KUKA KRL program: MyProgram_172().src

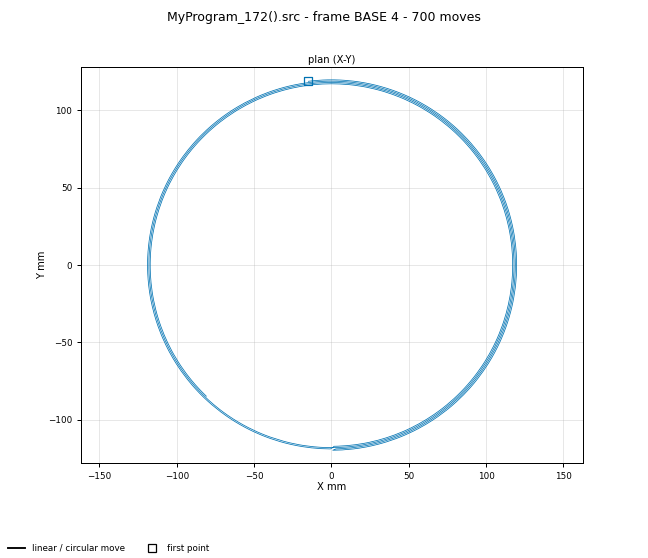
[picture p0: tool path of MyProgram_172().src in frame BASE 4, 700 of 700 moves have a stored position in this frame; points joined in program order, loops and branches not executed]
&ACCESS RVP
&REL 1
&PARAM TEMPLATE = C:\KRC\Roboter\Template\vorgabe
&PARAM EDITMASK = *
DEF MyProgram_172()
; ---- Setting reference (Base) ----
$BASE = BASE_DATA[4]

; --------------------------
; ---- Setting tool (TCP) ----
$TOOL = TOOL_DATA[3]
; --------------------------

$VEL.CP = VEL_APROX_PRINT
Startdeposition()
$VEL.CP = VEL_PRINT
LIN {X -14.9345,Y 118.8395,Z 128,A 91.9822,B 24.9419,C -1.7603,E1 24.9831,E2 354.1714} C_DIS
LIN {X -10.7622,Y 119.2891,Z 128,A 90.661,B 24.9398,C -1.7917,E1 24.9865,E2 355.4188} C_DIS
LIN {X -5.4739,Y 119.6487,Z 128,A 88.2073,B 24.9395,C -1.7964,E1 24.9934,E2 357.8622} C_DIS
LIN {X -2.3345,Y 119.7507,Z 128,A 85.9891,B 24.9416,C -1.7648,E1 24.9997,E2 360.1555} C_DIS
LIN {X 1.6856,Y 119.7625,Z 128,A 84.4618,B 24.9404,C -1.7828,E1 25.0039,E2 361.6401} C_DIS
LIN {X 5.7094,Y 119.6385,Z 128,A 82.6922,B 24.9399,C -1.7899,E1 25.0088,E2 363.3922} C_DIS
LIN {X 8.3372,Y 119.4831,Z 128,A 81.3395,B 24.9402,C -1.7857,E1 25.0126,E2 364.7544} C_DIS
LIN {X 14.2008,Y 118.9288,Z 128,A 78.7621,B 24.9395,C -1.7962,E1 25.0197,E2 367.3053} C_DIS
LIN {X 17.7257,Y 118.4559,Z 128,A 76.9686,B 24.9398,C -1.7916,E1 25.0247,E2 369.1083} C_DIS
LIN {X 21.7971,Y 117.7748,Z 128,A 74.9308,B 24.9401,C -1.788,E1 25.0303,E2 371.1525} C_DIS
LIN {X 25.2622,Y 117.0792,Z 128,A 73.1853,B 24.9403,C -1.7847,E1 25.0351,E2 372.9034} C_DIS
LIN {X 28.7779,Y 116.2654,Z 128,A 71.5409,B 24.9401,C -1.7875,E1 25.0395,E2 374.539} C_DIS
LIN {X 31.5389,Y 115.5467,Z 128,A 69.4789,B 24.9423,C -1.7548,E1 25.0453,E2 376.6751} C_DIS
LIN {X 35.9866,Y 114.2406,Z 128,A 67.9927,B 24.9402,C -1.7864,E1 25.049,E2 378.0836} C_DIS
LIN {X 39.7103,Y 112.9989,Z 128,A 65.8502,B 24.9411,C -1.7726,E1 25.0548,E2 380.2546} C_DIS
LIN {X 43.3363,Y 111.6596,Z 128,A 63.849,B 24.9417,C -1.7638,E1 25.06,E2 382.2724} C_DIS
LIN {X 47.456,Y 109.9717,Z 128,A 61.9358,B 24.9412,C -1.7715,E1 25.0649,E2 384.163} C_DIS
LIN {X 50.5894,Y 108.565,Z 128,A 60.3762,B 24.9411,C -1.7734,E1 25.0688,E2 385.714} C_DIS
LIN {X 54.0331,Y 106.8942,Z 128,A 58.4921,B 24.9414,C -1.7686,E1 25.0735,E2 387.6044} C_DIS
LIN {X 57.312,Y 105.1715,Z 128,A 56.7697,B 24.9414,C -1.7685,E1 25.0778,E2 389.3222} C_DIS
LIN {X 61.1307,Y 102.9987,Z 128,A 54.6582,B 24.9416,C -1.765,E1 25.0829,E2 391.4356} C_DIS
LIN {X 64.4896,Y 100.9297,Z 128,A 52.5109,B 24.9426,C -1.7498,E1 25.088,E2 393.6118} C_DIS
LIN {X 69.9469,Y 97.2281,Z 128,A 49.8821,B 24.9413,C -1.7692,E1 25.0939,E2 396.1859} C_DIS
LIN {X 73.3681,Y 94.6725,Z 128,A 47.6716,B 24.9421,C -1.7576,E1 25.0989,E2 398.4159} C_DIS
LIN {X 76.4144,Y 92.2308,Z 128,A 45.7857,B 24.9424,C -1.7531,E1 25.103,E2 400.3051} C_DIS
LIN {X 78.8231,Y 90.1808,Z 128,A 44.2978,B 24.9425,C -1.7513,E1 25.1061,E2 401.7914} C_DIS
LIN {X 81.4658,Y 87.8033,Z 128,A 42.4667,B 24.9432,C -1.7416,E1 25.11,E2 403.638} C_DIS
LIN {X 84.2691,Y 85.114,Z 128,A 40.7422,B 24.943,C -1.744,E1 25.1134,E2 405.3497} C_DIS
LIN {X 88.0039,Y 81.2472,Z 128,A 38.3973,B 24.9427,C -1.7491,E1 25.1179,E2 407.6724} C_DIS
LIN {X 90.3573,Y 78.621,Z 128,A 36.5475,B 24.9434,C -1.7374,E1 25.1213,E2 409.5416} C_DIS
LIN {X 93.9931,Y 74.2358,Z 128,A 33.8716,B 24.9437,C -1.7332,E1 25.1261,E2 412.2149} C_DIS
LIN {X 95.9007,Y 71.7548,Z 128,A 32.2244,B 24.9444,C -1.7223,E1 25.1289,E2 413.88} C_DIS
LIN {X 98.383,Y 68.3114,Z 128,A 30.2874,B 24.9444,C -1.7216,E1 25.132,E2 415.8092} C_DIS
LIN {X 100.4183,Y 65.2864,Z 128,A 28.4483,B 24.945,C -1.7125,E1 25.1348,E2 417.6608} C_DIS
LIN {X 102.3996,Y 62.1288,Z 128,A 26.0566,B 24.9472,C -1.6786,E1 25.1384,E2 420.1201} C_DIS
LIN {X 104.9804,Y 57.6644,Z 128,A 24.2184,B 24.9457,C -1.7019,E1 25.1408,E2 421.8939} C_DIS
LIN {X 106.7304,Y 54.3535,Z 128,A 22.5591,B 24.9457,C -1.7032,E1 25.1429,E2 423.5412} C_DIS
LIN {X 108.2379,Y 51.2896,Z 128,A 20.9731,B 24.9457,C -1.7009,E1 25.1449,E2 425.1243} C_DIS
LIN {X 109.6146,Y 48.2751,Z 128,A 19.0189,B 24.9472,C -1.6784,E1 25.1471,E2 427.1208} C_DIS
LIN {X 111.6551,Y 43.3476,Z 128,A 16.4448,B 24.9478,C -1.6698,E1 25.1498,E2 429.7011} C_DIS
LIN {X 112.8514,Y 40.1306,Z 128,A 15.3331,B 24.9464,C -1.6905,E1 25.1508,E2 430.7575} C_DIS
LIN {X 114.185,Y 36.1643,Z 128,A 13.0854,B 24.9476,C -1.6725,E1 25.1528,E2 433.0351} C_DIS
LIN {X 115.1759,Y 32.8666,Z 128,A 11.4964,B 24.9477,C -1.6702,E1 25.154,E2 434.6203} C_DIS
LIN {X 116.2749,Y 28.739,Z 128,A 9.4821,B 24.948,C -1.6653,E1 25.1554,E2 436.6346} C_DIS
LIN {X 117.0488,Y 25.4019,Z 128,A 7.9707,B 24.948,C -1.6664,E1 25.1563,E2 438.1348} C_DIS
LIN {X 117.6341,Y 22.5364,Z 128,A 6.5322,B 24.9484,C -1.66,E1 25.1571,E2 439.5799} C_DIS
LIN {X 118.2492,Y 19.0601,Z 128,A 4.6721,B 24.9492,C -1.6462,E1 25.158,E2 441.4616} C_DIS
LIN {X 119.1222,Y 12.4724,Z 128,A 2.0396,B 24.9482,C -1.6628,E1 25.1589,E2 444.0394} C_DIS
LIN {X 119.5152,Y 7.8623,Z 128,A -0.5581,B 24.9498,C -1.6367,E1 25.1595,E2 446.6832} C_DIS
LIN {X 119.7603,Y 1.8102,Z 128,A -3.0517,B 24.9492,C -1.6471,E1 25.1598,E2 449.1375} C_DIS
LIN {X 119.7522,Y -2.2507,Z 128,A -5.9251,B 24.9523,C -1.5952,E1 25.1597,E2 452.1161} C_DIS
LIN {X 119.5842,Y -6.7302,Z 128,A -7.1659,B 24.9501,C -1.6323,E1 25.1595,E2 453.2621} C_DIS
LIN {X 119.1569,Y -12.1411,Z 128,A -9.8149,B 24.9508,C -1.6211,E1 25.159,E2 455.9217} C_DIS
LIN {X 118.8189,Y -15.0932,Z 128,A -12.4654,B 24.9546,C -1.5566,E1 25.158,E2 458.7086} C_DIS
LIN {X 117.8363,Y -21.4551,Z 128,A -14.3715,B 24.9518,C -1.6036,E1 25.1571,E2 460.4928} C_DIS
LIN {X 117.3034,Y -24.199,Z 128,A -15.8035,B 24.9524,C -1.5946,E1 25.1563,E2 461.9377} C_DIS
LIN {X 116.6602,Y -27.131,Z 128,A -17.1963,B 24.9525,C -1.5921,E1 25.1555,E2 463.3283} C_DIS
LIN {X 115.915,Y -30.1577,Z 128,A -18.8453,B 24.9533,C -1.5795,E1 25.1543,E2 464.9974} C_DIS
LIN {X 114.8429,Y -34.0113,Z 128,A -20.6089,B 24.9532,C -1.5807,E1 25.153,E2 466.7481} C_DIS
LIN {X 113.9274,Y -36.9624,Z 128,A -22.1194,B 24.9536,C -1.5744,E1 25.1517,E2 468.2649} C_DIS
LIN {X 112.6185,Y -40.7776,Z 128,A -23.9811,B 24.9537,C -1.5716,E1 25.15,E2 470.1227} C_DIS
LIN {X 111.418,Y -43.9513,Z 128,A -25.65,B 24.9542,C -1.5643,E1 25.1483,E2 471.7995} C_DIS
LIN {X 109.366,Y -48.8355,Z 128,A -27.9679,B 24.954,C -1.567,E1 25.1458,E2 474.0982} C_DIS
LIN {X 107.4011,Y -53.0161,Z 128,A -30.0733,B 24.954,C -1.5654,E1 25.1433,E2 476.1962} C_DIS
LIN {X 105.5247,Y -56.6608,Z 128,A -32.7446,B 24.9564,C -1.5248,E1 25.1397,E2 478.9491} C_DIS
LIN {X 103.7146,Y -59.9083,Z 128,A -33.6102,B 24.9542,C -1.5641,E1 25.1386,E2 479.7175} C_DIS
LIN {X 101.3114,Y -63.8899,Z 128,A -36.3268,B 24.9559,C -1.5335,E1 25.1346,E2 482.4925} C_DIS
LIN {X 98.3282,Y -68.3902,Z 128,A -38.6382,B 24.9556,C -1.5394,E1 25.1311,E2 484.7785} C_DIS
LIN {X 94.2998,Y -73.8478,Z 128,A -42.0752,B 24.9567,C -1.521,E1 25.1253,E2 488.2423} C_DIS
LIN {X 92.1735,Y -76.4833,Z 128,A -44.2995,B 24.9585,C -1.4875,E1 25.1212,E2 490.5355} C_DIS
LIN {X 89.1898,Y -79.9427,Z 128,A -46.6277,B 24.9592,C -1.475,E1 25.1168,E2 492.8828} C_DIS
LIN {X 85.5452,Y -83.8326,Z 128,A -48.3712,B 24.9574,C -1.5074,E1 25.1136,E2 494.5425} C_DIS
LIN {X 80.5462,Y -88.6471,Z 128,A -52.2709,B 24.9594,C -1.4715,E1 25.1055,E2 498.5108} C_DIS
LIN {X 77.2653,Y -91.5206,Z 128,A -53.8492,B 24.9584,C -1.491,E1 25.1023,E2 500.0369} C_DIS
LIN {X 74.2886,Y -93.9514,Z 128,A -56.7192,B 24.9613,C -1.4379,E1 25.0958,E2 503.0217} C_DIS
LIN {X 68.7364,Y -98.0875,Z 128,A -58.7295,B 24.9583,C -1.4928,E1 25.0915,E2 504.8953} C_DIS
LIN {X 65.3681,Y -100.3649,Z 128,A -61.6332,B 24.961,C -1.4433,E1 25.0845,E2 507.9063} C_DIS
LIN {X 60.8442,Y -103.1681,Z 128,A -62.9572,B 24.958,C -1.4966,E1 25.0816,E2 509.1002} C_DIS
LIN {X 55.6149,Y -106.0787,Z 128,A -66.1813,B 24.9593,C -1.4741,E1 25.0736,E2 512.368} C_DIS
LIN {X 52.8498,Y -107.4835,Z 128,A -67.6815,B 24.9595,C -1.4708,E1 25.0699,E2 513.8719} C_DIS
LIN {X 47.3838,Y -110.0032,Z 128,A -70.4733,B 24.9595,C -1.4705,E1 25.0628,E2 516.6576} C_DIS
LIN {X 44.9683,Y -111.0115,Z 128,A -71.7797,B 24.9597,C -1.4661,E1 25.0594,E2 517.9713} C_DIS
LIN {X 41.9329,Y -112.1943,Z 128,A -74.48,B 24.9627,C -1.4105,E1 25.052,E2 520.7973} C_DIS
LIN {X 35.5057,Y -114.3897,Z 128,A -76.5649,B 24.96,C -1.4608,E1 25.0468,E2 522.7594} C_DIS
LIN {X 32.4814,Y -115.2851,Z 128,A -78.0718,B 24.9601,C -1.4592,E1 25.0427,E2 524.2676} C_DIS
LIN {X 29.6802,Y -116.0378,Z 128,A -79.4968,B 24.9603,C -1.456,E1 25.0389,E2 525.698} C_DIS
LIN {X 25.968,Y -116.9253,Z 128,A -81.4039,B 24.9606,C -1.4504,E1 25.0336,E2 527.6156} C_DIS
LIN {X 22.512,Y -117.6388,Z 128,A -83.6176,B 24.962,C -1.4246,E1 25.0274,E2 529.8878} C_DIS
LIN {X 18.0591,Y -118.4043,Z 128,A -85.6229,B 24.9617,C -1.4302,E1 25.0219,E2 531.878} C_DIS
LIN {X 14.2771,Y -118.9199,Z 128,A -86.9177,B 24.9604,C -1.4536,E1 25.0185,E2 533.1163} C_DIS
LIN {X 6.9052,Y -119.5745,Z 128,A -90.2911,B 24.9601,C -1.4595,E1 25.0092,E2 536.4739} C_DIS
LIN {X 0.8345,Y -119.7701,Z 128,A -93.2214,B 24.9602,C -1.4573,E1 25.001,E2 539.4087} C_DIS
Enddeposition()
LIN {X 0.8345,Y -119.7701,Z 128,A -93.2214,B 24.9602,C -1.4573,E1 25.001,E2 539.4087} C_DIS
Startdeposition()
$VEL.CP = VEL_PRINT
LIN {X 2.8953,Y -118.8882,Z 128,A -91.2381,B 24.9568,C -1.5184,E1 25.0069,E2 537.281} C_DIS
LIN {X 6.7932,Y -118.7278,Z 128,A -89.9008,B 24.9582,C -1.4939,E1 25.0105,E2 536.0023} C_DIS
LIN {X 12.3059,Y -118.2834,Z 128,A -87.272,B 24.9582,C -1.4936,E1 25.0178,E2 533.3757} C_DIS
LIN {X 15.4448,Y -117.9146,Z 128,A -85.7393,B 24.9582,C -1.495,E1 25.022,E2 531.8408} C_DIS
LIN {X 17.8503,Y -117.5749,Z 128,A -84.5445,B 24.958,C -1.497,E1 25.0253,E2 530.6425} C_DIS
LIN {X 23.2009,Y -116.6389,Z 128,A -81.8074,B 24.9576,C -1.5047,E1 25.0329,E2 527.8902} C_DIS
LIN {X 26.8874,Y -115.8424,Z 128,A -80.0744,B 24.9577,C -1.5025,E1 25.0376,E2 526.1647} C_DIS
LIN {X 30.6338,Y -114.9091,Z 128,A -78.1946,B 24.9575,C -1.5053,E1 25.0427,E2 524.281} C_DIS
LIN {X 33.7472,Y -114.0329,Z 128,A -76.6918,B 24.9575,C -1.5045,E1 25.0467,E2 522.7828} C_DIS
LIN {X 39.8877,Y -112.0341,Z 128,A -73.4398,B 24.957,C -1.515,E1 25.0554,E2 519.5121} C_DIS
LIN {X 43.5273,Y -110.6696,Z 128,A -71.7253,B 24.9573,C -1.5101,E1 25.0598,E2 517.813} C_DIS
LIN {X 46.4605,Y -109.471,Z 128,A -70.0701,B 24.9568,C -1.5185,E1 25.0641,E2 516.1419} C_DIS
LIN {X 49.1217,Y -108.3029,Z 128,A -68.4485,B 24.9561,C -1.5313,E1 25.0683,E2 514.4941} C_DIS
LIN {X 52.1685,Y -106.8707,Z 128,A -67.0331,B 24.9565,C -1.524,E1 25.0718,E2 513.0997} C_DIS
LIN {X 55.0721,Y -105.4021,Z 128,A -65.0797,B 24.9553,C -1.5453,E1 25.0768,E2 511.1014} C_DIS
LIN {X 58.7314,Y -103.4087,Z 128,A -63.5195,B 24.9563,C -1.5273,E1 25.0804,E2 509.5883} C_DIS
LIN {X 61.3868,Y -101.854,Z 128,A -61.5561,B 24.9548,C -1.5533,E1 25.0853,E2 507.5695} C_DIS
LIN {X 65.0646,Y -99.545,Z 128,A -60.0756,B 24.9563,C -1.5278,E1 25.0886,E2 506.154} C_DIS
LIN {X 67.6195,Y -97.8268,Z 128,A -58.7214,B 24.9564,C -1.5246,E1 25.0917,E2 504.812} C_DIS
LIN {X 72.6114,Y -94.1805,Z 128,A -55.5369,B 24.9555,C -1.5409,E1 25.0989,E2 501.6005} C_DIS
LIN {X 75.9071,Y -91.5451,Z 128,A -53.5631,B 24.9555,C -1.5426,E1 25.1031,E2 499.6301} C_DIS
LIN {X 78.1001,Y -89.6816,Z 128,A -51.9193,B 24.9545,C -1.5583,E1 25.1067,E2 497.9558} C_DIS
LIN {X 83.0665,Y -85.1049,Z 128,A -48.8714,B 24.9546,C -1.5561,E1 25.1128,E2 494.9257} C_DIS
LIN {X 85.6964,Y -82.4532,Z 128,A -47.4083,B 24.9553,C -1.5442,E1 25.1156,E2 493.4967} C_DIS
LIN {X 88.759,Y -79.1471,Z 128,A -44.6852,B 24.9534,C -1.5767,E1 25.1209,E2 490.709} C_DIS
LIN {X 90.922,Y -76.6547,Z 128,A -43.3461,B 24.9539,C -1.5686,E1 25.1232,E2 489.3952} C_DIS
LIN {X 93.1098,Y -73.9801,Z 128,A -41.8006,B 24.9539,C -1.5673,E1 25.1259,E2 487.86} C_DIS
LIN {X 96.737,Y -69.1689,Z 128,A -39.2022,B 24.9544,C -1.5604,E1 25.1302,E2 485.2902} C_DIS
LIN {X 98.2379,Y -67.0214,Z 128,A -37.4167,B 24.9527,C -1.5895,E1 25.1332,E2 483.4448} C_DIS
LIN {X 100.7124,Y -63.2414,Z 128,A -35.2399,B 24.9523,C -1.5958,E1 25.1364,E2 481.2641} C_DIS
LIN {X 103.0299,Y -59.3906,Z 128,A -33.3725,B 24.9528,C -1.5875,E1 25.139,E2 479.4259} C_DIS
LIN {X 105.3544,Y -55.1625,Z 128,A -30.927,B 24.952,C -1.6004,E1 25.1423,E2 476.9628} C_DIS
LIN {X 107.6576,Y -50.5209,Z 128,A -28.5211,B 24.9518,C -1.6035,E1 25.1452,E2 474.5625} C_DIS
LIN {X 109.3932,Y -46.6451,Z 128,A -26.3521,B 24.9511,C -1.6159,E1 25.1477,E2 472.3762} C_DIS
LIN {X 111.054,Y -42.5393,Z 128,A -24.3086,B 24.9509,C -1.6181,E1 25.1498,E2 470.3387} C_DIS
LIN {X 112.2755,Y -39.1998,Z 128,A -22.6928,B 24.9509,C -1.6187,E1 25.1513,E2 468.7306} C_DIS
LIN {X 113.4977,Y -35.5069,Z 128,A -20.8268,B 24.9506,C -1.6243,E1 25.1529,E2 466.862} C_DIS
LIN {X 114.4075,Y -32.4548,Z 128,A -19.3213,B 24.9504,C -1.6278,E1 25.154,E2 465.3569} C_DIS
LIN {X 115.2334,Y -29.3887,Z 128,A -17.7706,B 24.95,C -1.6337,E1 25.1551,E2 463.8011} C_DIS
LIN {X 116.1074,Y -25.7218,Z 128,A -15.9405,B 24.9496,C -1.6403,E1 25.1563,E2 461.9662} C_DIS
LIN {X 116.8616,Y -22.0444,Z 128,A -14.2309,B 24.9496,C -1.6413,E1 25.1572,E2 460.2643} C_DIS
LIN {X 117.8335,Y -16.0654,Z 128,A -11.1596,B 24.9485,C -1.6583,E1 25.1585,E2 457.1709} C_DIS
LIN {X 118.2758,Y -12.3783,Z 128,A -9.5565,B 24.9487,C -1.655,E1 25.159,E2 455.585} C_DIS
LIN {X 118.6721,Y -7.7074,Z 128,A -7.3093,B 24.9482,C -1.6618,E1 25.1595,E2 453.335} C_DIS
LIN {X 118.876,Y -3.3144,Z 128,A -5.0425,B 24.9474,C -1.6761,E1 25.1598,E2 451.0482} C_DIS
LIN {X 118.9205,Y 0.6044,Z 128,A -3.1956,B 24.9471,C -1.6802,E1 25.1598,E2 449.2025} C_DIS
LIN {X 118.8667,Y 3.6165,Z 128,A -1.6079,B 24.9464,C -1.6917,E1 25.1596,E2 447.5972} C_DIS
LIN {X 118.671,Y 7.7236,Z 128,A 0.2246,B 24.9464,C -1.6908,E1 25.1594,E2 445.7777} C_DIS
LIN {X 118.3124,Y 12.0286,Z 128,A 2.1778,B 24.9464,C -1.6912,E1 25.1589,E2 443.8351} C_DIS
LIN {X 117.7508,Y 16.6472,Z 128,A 4.5059,B 24.9457,C -1.7027,E1 25.158,E2 441.4937} C_DIS
LIN {X 117.1261,Y 20.5928,Z 128,A 6.365,B 24.9455,C -1.7056,E1 25.1572,E2 439.6387} C_DIS
LIN {X 116.5594,Y 23.5879,Z 128,A 7.8405,B 24.9452,C -1.7106,E1 25.1564,E2 438.1599} C_DIS
LIN {X 115.819,Y 26.9889,Z 128,A 9.5065,B 24.9449,C -1.7153,E1 25.1553,E2 436.4925} C_DIS
LIN {X 114.8458,Y 30.8681,Z 128,A 11.422,B 24.9445,C -1.7208,E1 25.154,E2 434.5752} C_DIS
LIN {X 113.7732,Y 34.6183,Z 128,A 13.2275,B 24.9444,C -1.7229,E1 25.1526,E2 432.7749} C_DIS
LIN {X 112.7393,Y 37.8453,Z 128,A 14.874,B 24.944,C -1.7286,E1 25.1511,E2 431.1244} C_DIS
LIN {X 111.527,Y 41.2829,Z 128,A 16.9498,B 24.9426,C -1.7495,E1 25.1491,E2 429.0109} C_DIS
LIN {X 110.3497,Y 44.3353,Z 128,A 18.1014,B 24.9437,C -1.7334,E1 25.148,E2 427.9036} C_DIS
LIN {X 108.8295,Y 47.9451,Z 128,A 20.1616,B 24.9428,C -1.7473,E1 25.1457,E2 425.8219} C_DIS
LIN {X 107.237,Y 51.4063,Z 128,A 21.7999,B 24.9431,C -1.743,E1 25.1437,E2 424.2025} C_DIS
LIN {X 105.9398,Y 54.0291,Z 128,A 23.2433,B 24.9427,C -1.7486,E1 25.1419,E2 422.7536} C_DIS
LIN {X 104.2675,Y 57.1925,Z 128,A 25.4236,B 24.9409,C -1.7756,E1 25.139,E2 420.521} C_DIS
LIN {X 102.4918,Y 60.3147,Z 128,A 26.725,B 24.942,C -1.7595,E1 25.1372,E2 419.2645} C_DIS
LIN {X 100.7835,Y 63.1275,Z 128,A 28.3407,B 24.9416,C -1.7652,E1 25.1348,E2 417.6436} C_DIS
LIN {X 98.755,Y 66.2577,Z 128,A 30.1557,B 24.9412,C -1.7707,E1 25.132,E2 415.8245} C_DIS
LIN {X 96.2669,Y 69.8237,Z 128,A 32.2134,B 24.941,C -1.7742,E1 25.1287,E2 413.7685} C_DIS
LIN {X 94.1897,Y 72.5994,Z 128,A 34.0169,B 24.9403,C -1.7848,E1 25.1256,E2 411.9486} C_DIS
LIN {X 90.6307,Y 76.9967,Z 128,A 36.53,B 24.9405,C -1.7811,E1 25.1212,E2 409.4559} C_DIS
LIN {X 88.4803,Y 79.4585,Z 128,A 38.1178,B 24.9403,C -1.7853,E1 25.1182,E2 407.8651} C_DIS
LIN {X 85.1795,Y 82.9895,Z 128,A 40.5633,B 24.9395,C -1.7961,E1 25.1135,E2 405.4048} C_DIS
LIN {X 82.6255,Y 85.5302,Z 128,A 42.0321,B 24.9401,C -1.7871,E1 25.1106,E2 403.9634} C_DIS
LIN {X 80.4784,Y 87.5535,Z 128,A 43.5573,B 24.9396,C -1.795,E1 25.1075,E2 402.4258} C_DIS
LIN {X 77.9739,Y 89.7918,Z 128,A 45.2458,B 24.9392,C -1.8016,E1 25.1039,E2 400.7285} C_DIS
LIN {X 74.9657,Y 92.3176,Z 128,A 47.0262,B 24.9392,C -1.7999,E1 25.1001,E2 398.9588} C_DIS
LIN {X 72.7007,Y 94.1117,Z 128,A 48.4539,B 24.939,C -1.8042,E1 25.0969,E2 397.5264} C_DIS
LIN {X 69.7825,Y 96.297,Z 128,A 50.2933,B 24.9385,C -1.8112,E1 25.0928,E2 395.6768} C_DIS
LIN {X 64.2278,Y 100.0858,Z 128,A 53.4071,B 24.9385,C -1.8106,E1 25.0856,E2 392.5749} C_DIS
LIN {X 61.242,Y 101.942,Z 128,A 55.116,B 24.9383,C -1.8139,E1 25.0815,E2 390.8637} C_DIS
LIN {X 57.6928,Y 103.9906,Z 128,A 57.2015,B 24.9378,C -1.8219,E1 25.0764,E2 388.7653} C_DIS
LIN {X 53.9956,Y 105.9569,Z 128,A 59.1105,B 24.9379,C -1.8196,E1 25.0717,E2 386.8672} C_DIS
LIN {X 50.427,Y 107.7013,Z 128,A 61.0237,B 24.9378,C -1.8219,E1 25.0669,E2 384.9535} C_DIS
LIN {X 46.8967,Y 109.2865,Z 128,A 62.857,B 24.9378,C -1.8225,E1 25.0622,E2 383.1231} C_DIS
LIN {X 42.8741,Y 110.9262,Z 128,A 65.0568,B 24.9373,C -1.8296,E1 25.0565,E2 380.9115} C_DIS
LIN {X 39.952,Y 112.0116,Z 128,A 66.5498,B 24.9372,C -1.8306,E1 25.0526,E2 379.4192} C_DIS
LIN {X 36.6887,Y 113.1209,Z 128,A 68.4007,B 24.9365,C -1.8408,E1 25.0476,E2 377.5476} C_DIS
LIN {X 30.1916,Y 115.027,Z 128,A 71.4659,B 24.937,C -1.8339,E1 25.0394,E2 374.5038} C_DIS
LIN {X 26.7632,Y 115.8711,Z 128,A 73.038,B 24.9373,C -1.829,E1 25.0352,E2 372.9457} C_DIS
LIN {X 23.4752,Y 116.5826,Z 128,A 74.7218,B 24.937,C -1.8326,E1 25.0306,E2 371.2554} C_DIS
LIN {X 19.8865,Y 117.2475,Z 128,A 76.4532,B 24.937,C -1.8321,E1 25.0258,E2 369.5271} C_DIS
LIN {X 16.75,Y 117.7362,Z 128,A 78.007,B 24.937,C -1.8336,E1 25.0215,E2 367.9711} C_DIS
LIN {X 13.6908,Y 118.1311,Z 128,A 79.6517,B 24.9365,C -1.8411,E1 25.0169,E2 366.3098} C_DIS
LIN {X 9.647,Y 118.5299,Z 128,A 81.4354,B 24.937,C -1.8334,E1 25.012,E2 364.5455} C_DIS
LIN {X 6.2648,Y 118.757,Z 128,A 83.1346,B 24.9368,C -1.8364,E1 25.0072,E2 362.8399} C_DIS
LIN {X 3.5328,Y 118.8693,Z 128,A 84.6064,B 24.9363,C -1.8433,E1 25.0031,E2 361.3521} C_DIS
LIN {X -2.1225,Y 118.9028,Z 128,A 87.0611,B 24.9372,C -1.8305,E1 24.9963,E2 358.9278} C_DIS
LIN {X -5.3436,Y 118.8019,Z 128,A 88.6163,B 24.9372,C -1.8301,E1 24.992,E2 357.3732} C_DIS
LIN {X -9.9585,Y 118.505,Z 128,A 90.8353,B 24.9373,C -1.8287,E1 24.9858,E2 355.1566} C_DIS
LIN {X -14.4655,Y 118.0404,Z 128,A 93.1902,B 24.9369,C -1.8352,E1 24.9792,E2 352.7849} C_DIS
LIN {X -17.7189,Y 117.5952,Z 128,A 94.6264,B 24.9374,C -1.8276,E1 24.9753,E2 351.3654} C_DIS
LIN {X -20.0668,Y 117.2174,Z 128,A 95.9288,B 24.937,C -1.8338,E1 24.9717,E2 350.0472} C_DIS
LIN {X -23.801,Y 116.5157,Z 128,A 97.6167,B 24.9375,C -1.8259,E1 24.9671,E2 348.376} C_DIS
LIN {X -26.8424,Y 115.8528,Z 128,A 99.0777,B 24.9377,C -1.8228,E1 24.9631,E2 346.9205} C_DIS
LIN {X -30.0884,Y 115.0535,Z 128,A 100.6609,B 24.9379,C -1.82,E1 24.9588,E2 345.3417} C_DIS
LIN {X -33.5329,Y 114.0965,Z 128,A 102.5958,B 24.9374,C -1.8275,E1 24.9536,E2 343.3858} C_DIS
LIN {X -37.7675,Y 112.7655,Z 128,A 104.995,B 24.9368,C -1.8365,E1 24.9472,E2 340.9609} C_DIS
LIN {X -41.0134,Y 111.626,Z 128,A 106.5558,B 24.9372,C -1.8301,E1 24.9431,E2 339.4123} C_DIS
LIN {X -45.7223,Y 109.7821,Z 128,A 108.7756,B 24.9381,C -1.8171,E1 24.9374,E2 337.2184} C_DIS
LIN {X -48.9642,Y 108.3739,Z 128,A 110.4611,B 24.9383,C -1.8138,E1 24.9331,E2 335.5367} C_DIS
LIN {X -56.0854,Y 104.868,Z 128,A 114.2258,B 24.9389,C -1.8048,E1 24.9238,E2 331.7832} C_DIS
LIN {X -60.9352,Y 102.125,Z 128,A 117.353,B 24.938,C -1.8193,E1 24.9161,E2 328.6124} C_DIS
LIN {X -63.8798,Y 100.3092,Z 128,A 118.7133,B 24.9391,C -1.8027,E1 24.913,E2 327.2871} C_DIS
LIN {X -67.1467,Y 98.1531,Z 128,A 121.0288,B 24.9381,C -1.8176,E1 24.9075,E2 324.9284} C_DIS
LIN {X -70.3204,Y 95.9032,Z 128,A 122.4423,B 24.9397,C -1.7938,E1 24.9045,E2 323.5667} C_DIS
LIN {X -72.843,Y 94.0021,Z 128,A 124.33,B 24.9388,C -1.8063,E1 24.9002,E2 321.6424} C_DIS
LIN {X -75.5923,Y 91.8067,Z 128,A 125.7074,B 24.94,C -1.7888,E1 24.8973,E2 320.3013} C_DIS
LIN {X -78.0818,Y 89.6975,Z 128,A 127.6243,B 24.9393,C -1.8001,E1 24.8932,E2 318.35} C_DIS
LIN {X -80.735,Y 87.3181,Z 128,A 128.8408,B 24.941,C -1.7745,E1 24.8908,E2 317.1896} C_DIS
LIN {X -84.8387,Y 83.336,Z 128,A 131.8205,B 24.9408,C -1.7774,E1 24.8848,E2 314.1904} C_DIS
LIN {X -87.002,Y 81.076,Z 128,A 133.6264,B 24.9402,C -1.7864,E1 24.8813,E2 312.3552} C_DIS
LIN {X -89.3075,Y 78.5284,Z 128,A 135.6609,B 24.9394,C -1.7984,E1 24.8775,E2 310.2829} C_DIS
LIN {X -92.6334,Y 74.5761,Z 128,A 137.5207,B 24.9416,C -1.7648,E1 24.8744,E2 308.4945} C_DIS
LIN {X -95.8128,Y 70.444,Z 128,A 139.9826,B 24.9422,C -1.7558,E1 24.8702,E2 306.0423} C_DIS
LIN {X -98.1595,Y 67.1373,Z 128,A 142.1479,B 24.942,C -1.7594,E1 24.8668,E2 303.8579} C_DIS
LIN {X -100.6825,Y 63.2893,Z 128,A 143.9033,B 24.9437,C -1.7335,E1 24.8642,E2 302.1553} C_DIS
LIN {X -103.2815,Y 58.9528,Z 128,A 146.0966,B 24.9448,C -1.7162,E1 24.8611,E2 299.9918} C_DIS
LIN {X -104.8822,Y 56.0591,Z 128,A 148.3085,B 24.9434,C -1.7374,E1 24.8581,E2 297.7176} C_DIS
LIN {X -106.7832,Y 52.3451,Z 128,A 150.24,B 24.944,C -1.7281,E1 24.8556,E2 295.798} C_DIS
LIN {X -109.0275,Y 47.4908,Z 128,A 152.7832,B 24.9446,C -1.7188,E1 24.8527,E2 293.263} C_DIS
LIN {X -110.4216,Y 44.1585,Z 128,A 154.6909,B 24.9446,C -1.7204,E1 24.8507,E2 291.3408} C_DIS
LIN {X -112.9098,Y 37.3392,Z 128,A 158.1235,B 24.9454,C -1.7067,E1 24.8475,E2 287.9215} C_DIS
LIN {X -113.9717,Y 33.9538,Z 128,A 159.8185,B 24.9458,C -1.7007,E1 24.8461,E2 286.2312} C_DIS
LIN {X -114.879,Y 30.7452,Z 128,A 161.9292,B 24.9448,C -1.7168,E1 24.8446,E2 284.0696} C_DIS
LIN {X -115.8564,Y 26.8266,Z 128,A 163.3574,B 24.9466,C -1.6887,E1 24.8437,E2 282.7001} C_DIS
LIN {X -116.6289,Y 23.2493,Z 128,A 165.2692,B 24.9466,C -1.6892,E1 24.8426,E2 280.7759} C_DIS
LIN {X -117.2972,Y 19.5892,Z 128,A 166.9465,B 24.9472,C -1.6785,E1 24.8418,E2 279.114} C_DIS
LIN {X -117.8729,Y 15.7667,Z 128,A 168.8275,B 24.9475,C -1.6732,E1 24.8411,E2 277.2344} C_DIS
LIN {X -118.264,Y 12.4904,Z 128,A 170.4435,B 24.9478,C -1.6691,E1 24.8405,E2 275.6185} C_DIS
LIN {X -118.6093,Y 8.6364,Z 128,A 172.3991,B 24.9479,C -1.6669,E1 24.8401,E2 273.6565} C_DIS
LIN {X -118.8076,Y 5.2104,Z 128,A 173.9314,B 24.9486,C -1.6564,E1 24.8399,E2 272.14} C_DIS
LIN {X -118.9026,Y 2.1331,Z 128,A 175.4673,B 24.9488,C -1.6538,E1 24.8398,E2 270.6011} C_DIS
LIN {X -118.9089,Y -1.7907,Z 128,A 177.4422,B 24.9489,C -1.6511,E1 24.8398,E2 268.6206} C_DIS
LIN {X -118.7971,Y -5.4544,Z 128,A 179.2482,B 24.9492,C -1.6471,E1 24.84,E2 266.8134} C_DIS
LIN {X -118.5481,Y -9.4203,Z 128,A -178.9518,B 24.9498,C -1.6361,E1 24.8404,E2 265.0289} C_DIS
LIN {X -118.2091,Y -13.0155,Z 128,A -177.0692,B 24.9498,C -1.6364,E1 24.8409,E2 263.134} C_DIS
LIN {X -117.7416,Y -16.7122,Z 128,A -175.3917,B 24.9505,C -1.6257,E1 24.8415,E2 261.4721} C_DIS
LIN {X -117.2296,Y -19.9937,Z 128,A -173.8845,B 24.951,C -1.6167,E1 24.8422,E2 259.9775} C_DIS
LIN {X -116.7,Y -22.8816,Z 128,A -172.2904,B 24.9508,C -1.6198,E1 24.8431,E2 258.3665} C_DIS
LIN {X -115.8726,Y -26.7569,Z 128,A -169.7086,B 24.9494,C -1.6425,E1 24.8447,E2 255.7154} C_DIS
LIN {X -114.6593,Y -31.5587,Z 128,A -168.362,B 24.9526,C -1.5908,E1 24.8456,E2 254.4841} C_DIS
LIN {X -113.3564,Y -35.9607,Z 128,A -165.6684,B 24.9518,C -1.6044,E1 24.8478,E2 251.7427} C_DIS
LIN {X -112.1181,Y -39.6484,Z 128,A -163.5809,B 24.9516,C -1.6079,E1 24.8497,E2 249.6351} C_DIS
LIN {X -110.2465,Y -44.5887,Z 128,A -161.3271,B 24.9528,C -1.5879,E1 24.852,E2 247.4162} C_DIS
LIN {X -109.0783,Y -47.3745,Z 128,A -159.8544,B 24.953,C -1.5844,E1 24.8536,E2 245.9437} C_DIS
LIN {X -106.8749,Y -52.1587,Z 128,A -157.2103,B 24.9531,C -1.5816,E1 24.8568,E2 243.2918} C_DIS
LIN {X -104.91,Y -56.005,Z 128,A -154.4984,B 24.9518,C -1.603,E1 24.8604,E2 240.5145} C_DIS
LIN {X -102.4915,Y -60.3152,Z 128,A -152.7723,B 24.9539,C -1.5683,E1 24.8627,E2 238.8622} C_DIS
LIN {X -100.4358,Y -63.6826,Z 128,A -150.8352,B 24.9541,C -1.5648,E1 24.8656,E2 236.9237} C_DIS
LIN {X -97.2172,Y -68.496,Z 128,A -147.985,B 24.9544,C -1.5602,E1 24.8701,E2 234.0702} C_DIS
LIN {X -93.0005,Y -74.1183,Z 128,A -144.6026,B 24.9549,C -1.5517,E1 24.8758,E2 230.6919} C_DIS
LIN {X -90.067,Y -77.6583,Z 128,A -142.333,B 24.9551,C -1.5488,E1 24.8799,E2 228.4187} C_DIS
LIN {X -87.7433,Y -80.2716,Z 128,A -140.5697,B 24.9551,C -1.5485,E1 24.8832,E2 226.6484} C_DIS
LIN {X -84.7811,Y -83.3943,Z 128,A -138.7582,B 24.956,C -1.5325,E1 24.8867,E2 224.8672} C_DIS
LIN {X -82.4675,Y -85.6826,Z 128,A -137.2865,B 24.9564,C -1.525,E1 24.8896,E2 223.4072} C_DIS
LIN {X -80.0537,Y -87.9432,Z 128,A -135.4181,B 24.9559,C -1.5337,E1 24.8935,E2 221.5104} C_DIS
LIN {X -77.1627,Y -90.4892,Z 128,A -133.7241,B 24.9565,C -1.523,E1 24.897,E2 219.8354} C_DIS
LIN {X -73.4624,Y -93.5189,Z 128,A -131.4018,B 24.9567,C -1.5194,E1 24.9021,E2 217.5129} C_DIS
LIN {X -71.6328,Y -94.9273,Z 128,A -129.5019,B 24.9549,C -1.5523,E1 24.9065,E2 215.5279} C_DIS
LIN {X -67.538,Y -97.8835,Z 128,A -127.6972,B 24.9567,C -1.5202,E1 24.9105,E2 213.7933} C_DIS
LIN {X -64.3296,Y -100.0205,Z 128,A -126.0068,B 24.9573,C -1.5099,E1 24.9144,E2 212.122} C_DIS
LIN {X -61.9604,Y -101.5054,Z 128,A -124.6231,B 24.9573,C -1.5094,E1 24.9177,E2 210.7349} C_DIS
LIN {X -59.3037,Y -103.0799,Z 128,A -123.0488,B 24.9573,C -1.5111,E1 24.9215,E2 209.152} C_DIS
LIN {X -55.7675,Y -105.0358,Z 128,A -121.1382,B 24.9575,C -1.5069,E1 24.9262,E2 207.2461} C_DIS
LIN {X -53.0195,Y -106.4489,Z 128,A -119.6668,B 24.9576,C -1.5042,E1 24.9298,E2 205.7771} C_DIS
LIN {X -50.2912,Y -107.7645,Z 128,A -118.2212,B 24.9577,C -1.5018,E1 24.9335,E2 204.3334} C_DIS
LIN {X -45.7755,Y -109.7597,Z 128,A -115.6843,B 24.9575,C -1.5063,E1 24.94,E2 201.7799} C_DIS
LIN {X -42.6927,Y -110.9959,Z 128,A -114.0724,B 24.9575,C -1.5053,E1 24.9442,E2 200.167} C_DIS
LIN {X -39.4635,Y -112.183,Z 128,A -112.2632,B 24.9572,C -1.5107,E1 24.949,E2 198.3413} C_DIS
LIN {X -33.0166,Y -114.2483,Z 128,A -109.1941,B 24.9579,C -1.4995,E1 24.9571,E2 195.2936} C_DIS
LIN {X -29.7606,Y -115.1378,Z 128,A -107.6074,B 24.958,C -1.4967,E1 24.9614,E2 193.711} C_DIS
LIN {X -26.3292,Y -115.9714,Z 128,A -105.8878,B 24.958,C -1.4967,E1 24.9661,E2 191.9893} C_DIS
LIN {X -22.5911,Y -116.7563,Z 128,A -104.1306,B 24.9583,C -1.4921,E1 24.9709,E2 190.2409} C_DIS
LIN {X -18.6279,Y -117.4546,Z 128,A -102.1036,B 24.9581,C -1.4955,E1 24.9765,E2 188.2039} C_DIS
LIN {X -13.0391,Y -118.2066,Z 128,A -99.3314,B 24.958,C -1.4976,E1 24.9842,E2 185.4248} C_DIS
LIN {X -9.0773,Y -118.5755,Z 128,A -97.5412,B 24.9583,C -1.4917,E1 24.9891,E2 183.6478} C_DIS
LIN {X -6.6936,Y -118.7333,Z 128,A -96.1853,B 24.9578,C -1.5012,E1 24.993,E2 182.269} C_DIS
LIN {X -0.6818,Y -118.9198,Z 128,A -93.4409,B 24.9582,C -1.4945,E1 25.0006,E2 179.5401} C_DIS
LIN {X -0.6818,Y -118.9198,Z 128,A -93.4409,B 24.9582,C -1.4945,E1 25.0006,E2 179.5401} C_DIS
Enddeposition()
LIN {X 0.8198,Y -118.067,Z 128,A -92.6855,B 24.9572,C -1.5109,E1 25.0028,E2 178.7459} C_DIS
Startdeposition()
$VEL.CP = VEL_PRINT
LIN {X -2.8079,Y -118.0384,Z 128,A -95.3031,B 24.9594,C -1.4714,E1 24.9952,E2 181.4571} C_DIS
LIN {X -7.3247,Y -117.8444,Z 128,A -97.3645,B 24.9591,C -1.4773,E1 24.9895,E2 183.5052} C_DIS
LIN {X -11.465,Y -117.5138,Z 128,A -99.4169,B 24.9592,C -1.4757,E1 24.9838,E2 185.5623} C_DIS
LIN {X -15.194,Y -117.0884,Z 128,A -101.16,B 24.959,C -1.4795,E1 24.979,E2 187.2975} C_DIS
LIN {X -17.6851,Y -116.7387,Z 128,A -102.564,B 24.9594,C -1.4716,E1 24.9751,E2 188.7214} C_DIS
LIN {X -20.908,Y -116.2042,Z 128,A -104.1342,B 24.9594,C -1.4728,E1 24.9707,E2 190.2903} C_DIS
LIN {X -24.0495,Y -115.5953,Z 128,A -105.5965,B 24.9591,C -1.4775,E1 24.9668,E2 191.7432} C_DIS
LIN {X -26.7451,Y -115.0012,Z 128,A -107.0017,B 24.9592,C -1.4752,E1 24.9629,E2 193.1555} C_DIS
LIN {X -30.5821,Y -114.041,Z 128,A -108.9259,B 24.9592,C -1.4761,E1 24.9577,E2 195.0804} C_DIS
LIN {X -39.4427,Y -111.2878,Z 128,A -113.1409,B 24.9583,C -1.4922,E1 24.9466,E2 199.2646} C_DIS
LIN {X -42.342,Y -110.2181,Z 128,A -114.8301,B 24.9587,C -1.4852,E1 24.9421,E2 200.974} C_DIS
LIN {X -45.14,Y -109.1027,Z 128,A -116.3396,B 24.9587,C -1.4846,E1 24.9382,E2 202.4883} C_DIS
LIN {X -48.236,Y -107.7679,Z 128,A -118.0625,B 24.9588,C -1.4826,E1 24.9338,E2 204.22} C_DIS
LIN {X -51.4162,Y -106.2875,Z 128,A -119.6844,B 24.9585,C -1.4882,E1 24.9297,E2 205.8328} C_DIS
LIN {X -53.7479,Y -105.1272,Z 128,A -120.9784,B 24.9585,C -1.4885,E1 24.9264,E2 207.1295} C_DIS
LIN {X -56.8989,Y -103.4579,Z 128,A -122.8817,B 24.9588,C -1.4833,E1 24.9217,E2 209.0506} C_DIS
LIN {X -60.2266,Y -101.5546,Z 128,A -124.545,B 24.9582,C -1.4945,E1 24.9178,E2 210.6921} C_DIS
LIN {X -63.2488,Y -99.7023,Z 128,A -126.242,B 24.958,C -1.4981,E1 24.9137,E2 212.3859} C_DIS
LIN {X -65.6031,Y -98.1697,Z 128,A -127.6489,B 24.958,C -1.4984,E1 24.9105,E2 213.7967} C_DIS
LIN {X -67.4094,Y -96.9357,Z 128,A -129.1572,B 24.9589,C -1.481,E1 24.9069,E2 215.3514} C_DIS
LIN {X -70.3226,Y -94.8462,Z 128,A -130.4625,B 24.9577,C -1.5027,E1 24.9041,E2 216.61} C_DIS
LIN {X -72.5651,Y -93.141,Z 128,A -132.2171,B 24.9585,C -1.4886,E1 24.9001,E2 218.4045} C_DIS
LIN {X -76.3914,Y -90.0276,Z 128,A -134.3385,B 24.9576,C -1.5048,E1 24.8956,E2 220.4954} C_DIS
LIN {X -79.3603,Y -87.4236,Z 128,A -136.519,B 24.958,C -1.4974,E1 24.891,E2 222.7022} C_DIS
LIN {X -83.0975,Y -83.8773,Z 128,A -138.6679,B 24.9569,C -1.5176,E1 24.8868,E2 224.812} C_DIS
LIN {X -85.2145,Y -81.7259,Z 128,A -140.463,B 24.9575,C -1.5068,E1 24.8832,E2 226.6406} C_DIS
LIN {X -87.8186,Y -78.9209,Z 128,A -142.1375,B 24.9568,C -1.5187,E1 24.8801,E2 228.294} C_DIS
LIN {X -89.943,Y -76.4907,Z 128,A -143.6118,B 24.9564,C -1.5262,E1 24.8775,E2 229.7572} C_DIS
LIN {X -92.0382,Y -73.9579,Z 128,A -145.4545,B 24.9567,C -1.5196,E1 24.8742,E2 231.6242} C_DIS
LIN {X -94.4093,Y -70.9044,Z 128,A -147.077,B 24.9559,C -1.5349,E1 24.8715,E2 233.218} C_DIS
LIN {X -96.178,Y -68.4862,Z 128,A -148.5681,B 24.9557,C -1.537,E1 24.869,E2 234.7114} C_DIS
LIN {X -98.474,Y -65.1418,Z 128,A -150.5682,B 24.9555,C -1.5408,E1 24.8659,E2 236.7124} C_DIS
LIN {X -100.4163,Y -62.108,Z 128,A -152.2581,B 24.9551,C -1.5478,E1 24.8634,E2 238.3942} C_DIS
LIN {X -101.8064,Y -59.8006,Z 128,A -154.3714,B 24.9568,C -1.5178,E1 24.8603,E2 240.5898} C_DIS
LIN {X -104.248,Y -55.4359,Z 128,A -156.1451,B 24.9549,C -1.5516,E1 24.858,E2 242.2925} C_DIS
LIN {X -105.8604,Y -52.2891,Z 128,A -158.0967,B 24.9552,C -1.5466,E1 24.8556,E2 244.2664} C_DIS
LIN {X -107.8771,Y -47.9937,Z 128,A -160.0617,B 24.954,C -1.5673,E1 24.8533,E2 246.193} C_DIS
LIN {X -108.8261,Y -45.7977,Z 128,A -161.2528,B 24.9539,C -1.5694,E1 24.852,E2 247.3856} C_DIS
LIN {X -110.0012,Y -42.8997,Z 128,A -162.9132,B 24.9539,C -1.568,E1 24.8503,E2 249.0587} C_DIS
LIN {X -111.1117,Y -39.9382,Z 128,A -164.3026,B 24.9533,C -1.5786,E1 24.849,E2 250.4307} C_DIS
LIN {X -112.1859,Y -36.8121,Z 128,A -166.0594,B 24.9533,C -1.5771,E1 24.8474,E2 252.201} C_DIS
LIN {X -113.3932,Y -32.9095,Z 128,A -168.894,B 24.9551,C -1.5483,E1 24.8451,E2 255.1208} C_DIS
LIN {X -114.8702,Y -27.3079,Z 128,A -170.7248,B 24.9522,C -1.5971,E1 24.844,E2 256.8457} C_DIS
LIN {X -116.153,Y -21.1928,Z 128,A -173.622,B 24.9513,C -1.6123,E1 24.8424,E2 259.7239} C_DIS
LIN {X -116.6803,Y -18.0627,Z 128,A -175.3512,B 24.9515,C -1.6094,E1 24.8415,E2 261.4703} C_DIS
LIN {X -117.093,Y -15.1588,Z 128,A -176.8309,B 24.9513,C -1.6116,E1 24.841,E2 262.9535} C_DIS
LIN {X -117.5088,Y -11.5192,Z 128,A -178.5607,B 24.9509,C -1.6193,E1 24.8405,E2 264.6754} C_DIS
LIN {X -117.6994,Y -9.3495,Z 128,A -179.6651,B 24.9508,C -1.6208,E1 24.8402,E2 265.7829} C_DIS
LIN {X -117.9115,Y -6.1308,Z 128,A 178.6169,B 24.9508,C -1.6196,E1 24.8399,E2 267.5141} C_DIS
LIN {X -118.0489,Y -2.2413,Z 128,A 176.8449,B 24.9502,C -1.6305,E1 24.8398,E2 269.2706} C_DIS
LIN {X -118.0649,Y 1.2337,Z 128,A 175.1602,B 24.9498,C -1.6361,E1 24.8398,E2 270.9523} C_DIS
LIN {X -118.0067,Y 3.8792,Z 128,A 173.7332,B 24.9499,C -1.6344,E1 24.8399,E2 272.3918} C_DIS
LIN {X -117.8151,Y 7.7586,Z 128,A 171.9378,B 24.9493,C -1.6442,E1 24.8402,E2 274.1746} C_DIS
LIN {X -117.5532,Y 11.0374,Z 128,A 170.3264,B 24.9491,C -1.6488,E1 24.8406,E2 275.7847} C_DIS
LIN {X -117.2075,Y 14.256,Z 128,A 168.6241,B 24.9491,C -1.6486,E1 24.8411,E2 277.4979} C_DIS
LIN {X -116.6809,Y 18.0586,Z 128,A 166.8101,B 24.9486,C -1.6567,E1 24.8419,E2 279.3033} C_DIS
LIN {X -116.044,Y 21.7864,Z 128,A 164.9394,B 24.9483,C -1.6611,E1 24.8428,E2 281.1745} C_DIS
LIN {X -115.3104,Y 25.3793,Z 128,A 163.05,B 24.9483,C -1.6624,E1 24.8439,E2 283.072} C_DIS
LIN {X -114.385,Y 29.2683,Z 128,A 161.2251,B 24.9475,C -1.6734,E1 24.8451,E2 284.8815} C_DIS
LIN {X -113.5612,Y 32.3177,Z 128,A 159.6978,B 24.9472,C -1.6785,E1 24.8463,E2 286.4054} C_DIS
LIN {X -112.732,Y 35.1008,Z 128,A 158.2831,B 24.9469,C -1.6828,E1 24.8474,E2 287.818} C_DIS
LIN {X -111.4684,Y 38.9278,Z 128,A 156.1412,B 24.947,C -1.6813,E1 24.8494,E2 289.9757} C_DIS
LIN {X -110.2173,Y 42.344,Z 128,A 154.6171,B 24.9461,C -1.6967,E1 24.8508,E2 291.4716} C_DIS
LIN {X -109.2745,Y 44.7179,Z 128,A 153.3285,B 24.9459,C -1.6985,E1 24.8522,E2 292.763} C_DIS
LIN {X -107.6572,Y 48.4819,Z 128,A 151.268,B 24.9457,C -1.7017,E1 24.8545,E2 294.8274} C_DIS
LIN {X -105.7954,Y 52.4203,Z 128,A 149.1699,B 24.9453,C -1.7087,E1 24.857,E2 296.9201} C_DIS
LIN {X -104.4227,Y 55.1041,Z 128,A 147.698,B 24.945,C -1.7127,E1 24.8589,E2 298.3903} C_DIS
LIN {X -102.6391,Y 58.3614,Z 128,A 145.6109,B 24.9454,C -1.7063,E1 24.8618,E2 300.5037} C_DIS
LIN {X -99.6765,Y 63.2889,Z 128,A 142.8918,B 24.9447,C -1.7172,E1 24.8658,E2 303.2106} C_DIS
LIN {X -97.5907,Y 66.4584,Z 128,A 141.2273,B 24.9439,C -1.7297,E1 24.8683,E2 304.8536} C_DIS
LIN {X -95.7732,Y 69.0536,Z 128,A 139.6184,B 24.9439,C -1.731,E1 24.8709,E2 306.4673} C_DIS
LIN {X -93.4635,Y 72.1467,Z 128,A 137.7998,B 24.9434,C -1.7384,E1 24.874,E2 308.2769} C_DIS
LIN {X -90.4139,Y 75.9359,Z 128,A 135.5009,B 24.9428,C -1.7472,E1 24.878,E2 310.5657} C_DIS
LIN {X -88.257,Y 78.4311,Z 128,A 133.6826,B 24.9431,C -1.7423,E1 24.8814,E2 312.4038} C_DIS
LIN {X -85.8684,Y 81.0384,Z 128,A 132.0599,B 24.9426,C -1.7505,E1 24.8845,E2 314.0141} C_DIS
LIN {X -81.9614,Y 84.9875,Z 128,A 129.4202,B 24.942,C -1.7594,E1 24.8897,E2 316.6436} C_DIS
LIN {X -79.5981,Y 87.2054,Z 128,A 127.6818,B 24.9422,C -1.7562,E1 24.8933,E2 318.3968} C_DIS
LIN {X -76.4907,Y 89.943,Z 128,A 125.811,B 24.9415,C -1.7666,E1 24.8972,E2 320.2501} C_DIS
LIN {X -73.5861,Y 92.3357,Z 128,A 124.1145,B 24.9409,C -1.7761,E1 24.9008,E2 321.9305} C_DIS
LIN {X -71.35,Y 94.0746,Z 128,A 122.4894,B 24.9414,C -1.7685,E1 24.9045,E2 323.5796} C_DIS
LIN {X -68.5282,Y 96.148,Z 128,A 120.7953,B 24.9411,C -1.7723,E1 24.9083,E2 325.2706} C_DIS
LIN {X -65.775,Y 98.0534,Z 128,A 119.1196,B 24.9411,C -1.7733,E1 24.9122,E2 326.9494} C_DIS
LIN {X -60.4162,Y 101.4426,Z 128,A 116.3427,B 24.9398,C -1.7919,E1 24.9187,E2 329.691} C_DIS
LIN {X -57.7609,Y 102.9771,Z 128,A 114.6077,B 24.9403,C -1.7841,E1 24.9229,E2 331.4496} C_DIS
LIN {X -54.4349,Y 104.7751,Z 128,A 112.551,B 24.9408,C -1.7777,E1 24.9281,E2 333.5271} C_DIS
LIN {X -49.9686,Y 106.9753,Z 128,A 110.3074,B 24.94,C -1.7889,E1 24.9337,E2 335.7499} C_DIS
LIN {X -46.7714,Y 108.4122,Z 128,A 108.7276,B 24.9395,C -1.7966,E1 24.9377,E2 337.3151} C_DIS
LIN {X -41.7881,Y 110.4279,Z 128,A 105.4548,B 24.9412,C -1.7719,E1 24.9464,E2 340.6537} C_DIS
LIN {X -37.605,Y 111.9216,Z 128,A 103.9106,B 24.9392,C -1.8007,E1 24.9503,E2 342.1324} C_DIS
LIN {X -32.0099,Y 113.6484,Z 128,A 101.1554,B 24.9388,C -1.8076,E1 24.9576,E2 344.8759} C_DIS
LIN {X -29.357,Y 114.3623,Z 128,A 99.7075,B 24.939,C -1.804,E1 24.9615,E2 346.3346} C_DIS
LIN {X -26.2163,Y 115.1234,Z 128,A 98.2354,B 24.9386,C -1.8096,E1 24.9655,E2 347.7952} C_DIS
LIN {X -23.4983,Y 115.7085,Z 128,A 96.7276,B 24.939,C -1.8039,E1 24.9697,E2 349.3184} C_DIS
LIN {X -20.3379,Y 116.3067,Z 128,A 95.2998,B 24.9385,C -1.8109,E1 24.9735,E2 350.7311} C_DIS
LIN {X -17.1543,Y 116.8186,Z 128,A 93.75,B 24.9385,C -1.8126,E1 24.9778,E2 352.2781} C_DIS
LIN {X -14.6599,Y 117.1576,Z 128,A 92.2749,B 24.9391,C -1.8023,E1 24.982,E2 353.7788} C_DIS
LIN {X -10.1796,Y 117.6324,Z 128,A 90.221,B 24.9386,C -1.8092,E1 24.9876,E2 355.8175} C_DIS
LIN {X -6.4575,Y 117.8934,Z 128,A 88.4727,B 24.9384,C -1.8127,E1 24.9925,E2 357.558} C_DIS
LIN {X -2.8479,Y 118.0377,Z 128,A 86.7571,B 24.9383,C -1.8148,E1 24.9973,E2 359.2689} C_DIS
LIN {X -0.2089,Y 118.0711,Z 128,A 85.4529,B 24.9383,C -1.8141,E1 25.0009,E2 360.5749} C_DIS
LIN {X 2.9909,Y 118.0339,Z 128,A 83.9219,B 24.9383,C -1.8153,E1 25.0052,E2 362.1028} C_DIS
LIN {X 6.4834,Y 117.892,Z 128,A 82.1368,B 24.9385,C -1.8114,E1 25.0102,E2 363.8965} C_DIS
LIN {X 9.8505,Y 117.6593,Z 128,A 80.4339,B 24.9387,C -1.8085,E1 25.0149,E2 365.6056} C_DIS
LIN {X 13.1808,Y 117.3334,Z 128,A 78.9626,B 24.9383,C -1.815,E1 25.019,E2 367.0605} C_DIS
LIN {X 15.6888,Y 117.0243,Z 128,A 77.7095,B 24.9383,C -1.8135,E1 25.0225,E2 368.316} C_DIS
LIN {X 19.4681,Y 116.4541,Z 128,A 75.8068,B 24.9385,C -1.8108,E1 25.0277,E2 370.2233} C_DIS
LIN {X 22.3811,Y 115.9295,Z 128,A 74.3939,B 24.9385,C -1.8113,E1 25.0316,E2 371.6335} C_DIS
LIN {X 26.0775,Y 115.1555,Z 128,A 72.4863,B 24.9388,C -1.807,E1 25.0368,E2 373.5488} C_DIS
LIN {X 29.4241,Y 114.345,Z 128,A 69.6611,B 24.9423,C -1.7546,E1 25.0448,E2 376.4935} C_DIS
LIN {X 36.3633,Y 112.3311,Z 128,A 67.7524,B 24.9377,C -1.8234,E1 25.0494,E2 378.236} C_DIS
LIN {X 39.4713,Y 111.2777,Z 128,A 65.7015,B 24.9392,C -1.8012,E1 25.055,E2 380.3355} C_DIS
LIN {X 43.1022,Y 109.9216,Z 128,A 63.8327,B 24.9392,C -1.7999,E1 25.0598,E2 382.2033} C_DIS
LIN {X 46.0189,Y 108.7329,Z 128,A 62.3825,B 24.9392,C -1.8018,E1 25.0636,E2 383.6455} C_DIS
LIN {X 48.8307,Y 107.5,Z 128,A 60.7935,B 24.9396,C -1.7955,E1 25.0676,E2 385.2455} C_DIS
LIN {X 52.7909,Y 105.6117,Z 128,A 58.6548,B 24.9398,C -1.7924,E1 25.073,E2 387.3859} C_DIS
LIN {X 56.2445,Y 103.8129,Z 128,A 56.8382,B 24.9398,C -1.7932,E1 25.0775,E2 389.1954} C_DIS
LIN {X 59.0451,Y 102.2462,Z 128,A 55.406,B 24.9395,C -1.7967,E1 25.0809,E2 390.6151} C_DIS
LIN {X 62.0056,Y 100.4803,Z 128,A 53.7568,B 24.9395,C -1.7952,E1 25.0849,E2 392.2627} C_DIS
LIN {X 64.0905,Y 99.162,Z 128,A 51.5149,B 24.9429,C -1.7455,E1 25.0904,E2 394.6148} C_DIS
LIN {X 69.1662,Y 95.6928,Z 128,A 49.557,B 24.9401,C -1.7873,E1 25.0946,E2 396.467} C_DIS
LIN {X 71.539,Y 93.9317,Z 128,A 48.0907,B 24.9404,C -1.7832,E1 25.0979,E2 397.9377} C_DIS
LIN {X 74.232,Y 91.816,Z 128,A 46.3726,B 24.9408,C -1.7775,E1 25.1016,E2 399.6628} C_DIS
LIN {X 77.4169,Y 89.1476,Z 128,A 44.3571,B 24.941,C -1.7736,E1 25.1059,E2 401.6797} C_DIS
LIN {X 80.1774,Y 86.6739,Z 128,A 42.5105,B 24.9414,C -1.7677,E1 25.1097,E2 403.5329} C_DIS
LIN {X 83.0565,Y 83.9177,Z 128,A 40.8351,B 24.9409,C -1.7757,E1 25.113,E2 405.1824} C_DIS
LIN {X 85.0641,Y 81.882,Z 128,A 39.319,B 24.9415,C -1.7666,E1 25.116,E2 406.7135} C_DIS
LIN {X 87.5882,Y 79.1782,Z 128,A 37.4539,B 24.942,C -1.7592,E1 25.1196,E2 408.5878} C_DIS
LIN {X 89.8875,Y 76.5558,Z 128,A 34.8382,B 24.9451,C -1.7122,E1 25.1245,E2 411.3024} C_DIS
LIN {X 93.8737,Y 71.6144,Z 128,A 32.8393,B 24.9423,C -1.7552,E1 25.1277,E2 413.1906} C_DIS
LIN {X 96.281,Y 68.3419,Z 128,A 30.9223,B 24.9424,C -1.7528,E1 25.1309,E2 415.104} C_DIS
LIN {X 98.2429,Y 65.4924,Z 128,A 29.257,B 24.9427,C -1.749,E1 25.1335,E2 416.7699} C_DIS
LIN {X 99.5193,Y 63.5338,Z 128,A 28.0856,B 24.943,C -1.7443,E1 25.1353,E2 417.9465} C_DIS
LIN {X 100.9603,Y 61.2176,Z 128,A 26.6693,B 24.9435,C -1.7364,E1 25.1373,E2 419.3744} C_DIS
LIN {X 102.5865,Y 58.453,Z 128,A 25.1076,B 24.9438,C -1.7319,E1 25.1395,E2 420.9385} C_DIS
LIN {X 104.4163,Y 55.1164,Z 128,A 23.3278,B 24.9439,C -1.7299,E1 25.1419,E2 422.7136} C_DIS
LIN {X 106.15,Y 51.7024,Z 128,A 21.545,B 24.944,C -1.7282,E1 25.1441,E2 424.491} C_DIS
LIN {X 107.2638,Y 49.3489,Z 128,A 20.3128,B 24.9442,C -1.7261,E1 25.1456,E2 425.7215} C_DIS
LIN {X 108.2617,Y 47.1165,Z 128,A 18.967,B 24.9449,C -1.7151,E1 25.1471,E2 427.086} C_DIS
LIN {X 109.5947,Y 43.9312,Z 128,A 16.6103,B 24.9472,C -1.6778,E1 25.1496,E2 429.5176} C_DIS
LIN {X 111.3941,Y 39.1397,Z 128,A 15.2538,B 24.9443,C -1.724,E1 25.1508,E2 430.7574} C_DIS
LIN {X 112.7614,Y 35.0061,Z 128,A 13.0132,B 24.9451,C -1.7114,E1 25.1528,E2 433.0151} C_DIS
LIN {X 113.4939,Y 32.5553,Z 128,A 11.5314,B 24.9461,C -1.696,E1 25.154,E2 434.5247} C_DIS
LIN {X 114.3328,Y 29.4716,Z 128,A 10.0716,B 24.9461,C -1.6956,E1 25.155,E2 435.9772} C_DIS
LIN {X 115.0804,Y 26.4026,Z 128,A 8.5135,B 24.9465,C -1.6896,E1 25.156,E2 437.5403} C_DIS
LIN {X 115.7637,Y 23.2294,Z 128,A 7.0026,B 24.9466,C -1.6877,E1 25.1569,E2 439.047} C_DIS
LIN {X 116.4044,Y 19.7651,Z 128,A 5.2463,B 24.9471,C -1.68,E1 25.1577,E2 440.811} C_DIS
LIN {X 116.9199,Y 16.4413,Z 128,A 3.6319,B 24.9474,C -1.6756,E1 25.1584,E2 442.4263} C_DIS
LIN {X 117.3876,Y 12.6834,Z 128,A 1.8321,B 24.9476,C -1.6715,E1 25.159,E2 444.2252} C_DIS
LIN {X 117.6988,Y 9.3566,Z 128,A 0.1904,B 24.948,C -1.6653,E1 25.1594,E2 445.8717} C_DIS
LIN {X 117.9435,Y 5.4826,Z 128,A -1.5485,B 24.948,C -1.6662,E1 25.1596,E2 447.5983} C_DIS
LIN {X 118.0351,Y 2.9516,Z 128,A -3.0692,B 24.9491,C -1.6481,E1 25.1598,E2 449.1526} C_DIS
LIN {X 118.0665,Y -0.9766,Z 128,A -4.7394,B 24.9488,C -1.6532,E1 25.1598,E2 450.8007} C_DIS
LIN {X 117.9901,Y -4.3898,Z 128,A -6.4019,B 24.9491,C -1.6475,E1 25.1596,E2 452.4668} C_DIS
LIN {X 117.8041,Y -7.9215,Z 128,A -8.1687,B 24.9496,C -1.6395,E1 25.1593,E2 454.2421} C_DIS
LIN {X 117.5653,Y -10.9071,Z 128,A -9.6143,B 24.9499,C -1.6351,E1 25.159,E2 455.6895} C_DIS
LIN {X 117.213,Y -14.2093,Z 128,A -11.1,B 24.9499,C -1.6359,E1 25.1585,E2 457.1645} C_DIS
LIN {X 116.8331,Y -17.0523,Z 128,A -12.7937,B 24.951,C -1.6167,E1 25.1579,E2 458.8933} C_DIS
LIN {X 116.0749,Y -21.6257,Z 128,A -14.7432,B 24.9506,C -1.6239,E1 25.1569,E2 460.8146} C_DIS
LIN {X 115.4494,Y -24.7421,Z 128,A -16.4127,B 24.9513,C -1.6127,E1 25.156,E2 462.5006} C_DIS
LIN {X 114.5124,Y -28.7726,Z 128,A -18.2487,B 24.9512,C -1.6145,E1 25.1548,E2 464.3217} C_DIS
LIN {X 113.5527,Y -32.3474,Z 128,A -20.0147,B 24.9514,C -1.6102,E1 25.1535,E2 466.0877} C_DIS
LIN {X 112.7473,Y -35.0514,Z 128,A -21.4327,B 24.9518,C -1.6035,E1 25.1523,E2 467.5135} C_DIS
LIN {X 111.6942,Y -38.2792,Z 128,A -23.0385,B 24.952,C -1.6003,E1 25.1509,E2 469.1179} C_DIS
LIN {X 110.8658,Y -40.6121,Z 128,A -24.3546,B 24.9526,C -1.591,E1 25.1496,E2 470.4484} C_DIS
LIN {X 109.6239,Y -43.8595,Z 128,A -25.917,B 24.9526,C -1.5917,E1 25.1481,E2 472.0006} C_DIS
LIN {X 108.6577,Y -46.1973,Z 128,A -27.326,B 24.9533,C -1.5792,E1 25.1465,E2 473.4313} C_DIS
LIN {X 105.8559,Y -52.2983,Z 128,A -30.5182,B 24.9537,C -1.5724,E1 25.1427,E2 476.6223} C_DIS
LIN {X 103.8303,Y -56.2124,Z 128,A -32.5398,B 24.9537,C -1.5716,E1 25.1401,E2 478.6351} C_DIS
LIN {X 102.0749,Y -59.3433,Z 128,A -34.3863,B 24.9543,C -1.5614,E1 25.1375,E2 480.4961} C_DIS
LIN {X 99.8387,Y -63.0327,Z 128,A -36.3399,B 24.9543,C -1.562,E1 25.1347,E2 482.4383} C_DIS
LIN {X 96.3455,Y -68.2515,Z 128,A -39.2062,B 24.9543,C -1.562,E1 25.1303,E2 485.2902} C_DIS
LIN {X 94.7828,Y -70.4065,Z 128,A -40.5722,B 24.9547,C -1.5549,E1 25.128,E2 486.6666} C_DIS
LIN {X 93.1001,Y -72.6183,Z 128,A -42.1717,B 24.9556,C -1.5392,E1 25.1252,E2 488.2955} C_DIS
LIN {X 90.6596,Y -75.6402,Z 128,A -43.8615,B 24.9554,C -1.5435,E1 25.1222,E2 489.9673} C_DIS
LIN {X 88.3283,Y -78.3515,Z 128,A -45.6978,B 24.9559,C -1.5341,E1 25.1188,E2 491.8175} C_DIS
LIN {X 86.0673,Y -80.8269,Z 128,A -47.226,B 24.9559,C -1.5347,E1 25.1159,E2 493.3377} C_DIS
LIN {X 83.9413,Y -83.0326,Z 128,A -48.7022,B 24.9561,C -1.5315,E1 25.113,E2 494.8152} C_DIS
LIN {X 81.6762,Y -85.2625,Z 128,A -50.3606,B 24.9566,C -1.5222,E1 25.1097,E2 496.4885} C_DIS
LIN {X 78.9628,Y -87.7811,Z 128,A -52.0488,B 24.9566,C -1.5231,E1 25.1062,E2 498.1679} C_DIS
LIN {X 76.493,Y -89.941,Z 128,A -53.6065,B 24.9566,C -1.521,E1 25.1029,E2 499.7243} C_DIS
LIN {X 73.6189,Y -92.3098,Z 128,A -55.4623,B 24.957,C -1.5147,E1 25.0989,E2 501.5881} C_DIS
LIN {X 70.8974,Y -94.4146,Z 128,A -57.2631,B 24.9576,C -1.5049,E1 25.0949,E2 503.4054} C_DIS
LIN {X 67.4838,Y -96.884,Z 128,A -59.1961,B 24.9576,C -1.5059,E1 25.0905,E2 505.3294} C_DIS
LIN {X 64.6611,Y -98.791,Z 128,A -60.9436,B 24.958,C -1.4981,E1 25.0864,E2 507.0894} C_DIS
LIN {X 61.1049,Y -101.0287,Z 128,A -62.792,B 24.9577,C -1.5032,E1 25.082,E2 508.92} C_DIS
LIN {X 57.9385,Y -102.8779,Z 128,A -64.5712,B 24.9579,C -1.4999,E1 25.0777,E2 510.7016} C_DIS
LIN {X 54.5293,Y -104.7255,Z 128,A -66.3409,B 24.9577,C -1.5019,E1 25.0734,E2 512.4616} C_DIS
LIN {X 50.2689,Y -106.8355,Z 128,A -68.7746,B 24.9583,C -1.4922,E1 25.0672,E2 514.9118} C_DIS
LIN {X 47.0902,Y -108.2732,Z 128,A -70.5178,B 24.9586,C -1.4872,E1 25.0628,E2 516.6623} C_DIS
LIN {X 44.0767,Y -109.5355,Z 128,A -71.9378,B 24.9583,C -1.4926,E1 25.0591,E2 518.0663} C_DIS
LIN {X 41.5671,Y -110.5115,Z 128,A -73.417,B 24.9588,C -1.4828,E1 25.0552,E2 519.5656} C_DIS
LIN {X 37.7642,Y -111.8679,Z 128,A -75.423,B 24.9591,C -1.4781,E1 25.0499,E2 521.5787} C_DIS
LIN {X 34.4644,Y -112.9294,Z 128,A -76.8838,B 24.9586,C -1.4863,E1 25.0461,E2 523.0174} C_DIS
LIN {X 31.1206,Y -113.8955,Z 128,A -78.6676,B 24.959,C -1.4801,E1 25.0413,E2 524.813} C_DIS
LIN {X 28.0573,Y -114.6881,Z 128,A -80.1391,B 24.9589,C -1.4815,E1 25.0373,E2 526.279} C_DIS
LIN {X 24.7792,Y -115.4413,Z 128,A -81.7618,B 24.9589,C -1.4804,E1 25.0329,E2 527.9022} C_DIS
LIN {X 19.566,Y -116.4377,Z 128,A -84.0398,B 24.9583,C -1.4919,E1 25.0267,E2 530.1503} C_DIS
LIN {X 15.7835,Y -117.012,Z 128,A -86.38,B 24.9596,C -1.4684,E1 25.0201,E2 532.5439} C_DIS
LIN {X 11.8996,Y -117.4696,Z 128,A -88.2247,B 24.9596,C -1.4697,E1 25.015,E2 534.3843} C_DIS
LIN {X 8.9403,Y -117.7321,Z 128,A -89.5704,B 24.9593,C -1.4734,E1 25.0113,E2 535.7207} C_DIS
LIN {X 4.8617,Y -117.9702,Z 128,A -91.5318,B 24.9593,C -1.4735,E1 25.0058,E2 537.681} C_DIS
LIN {X 0.8198,Y -118.067,Z 128,A -92.6832,B 24.9573,C -1.5099,E1 25.0028,E2 538.7459} C_DIS
Enddeposition()
LIN {X 0.8198,Y -118.067,Z 128,A -92.6832,B 24.9573,C -1.5099,E1 25.0028,E2 538.7459} C_DIS
Startdeposition()
$VEL.CP = VEL_PRINT
LIN {X 1.6898,Y -117.2073,Z 128,A -92.4843,B 24.957,C -1.5145,E1 25.0034,E2 538.5363} C_DIS
LIN {X 4.2995,Y -117.1418,Z 128,A -91.1401,B 24.9568,C -1.518,E1 25.0072,E2 537.1841} C_DIS
LIN {X 7.4408,Y -116.983,Z 128,A -89.606,B 24.9568,C -1.5185,E1 25.0114,E2 535.6494} C_DIS
LIN {X 10.0436,Y -116.7896,Z 128,A -88.3282,B 24.9568,C -1.5192,E1 25.015,E2 534.3705} C_DIS
LIN {X 13.1744,Y -116.4767,Z 128,A -86.7955,B 24.9568,C -1.5198,E1 25.0193,E2 532.8373} C_DIS
LIN {X 15.765,Y -116.1557,Z 128,A -85.4283,B 24.9564,C -1.5249,E1 25.0231,E2 531.4594} C_DIS
LIN {X 18.8534,Y -115.6934,Z 128,A -84.0991,B 24.9569,C -1.5169,E1 25.0267,E2 530.1503} C_DIS
LIN {X 21.4275,Y -115.2455,Z 128,A -82.5843,B 24.9562,C -1.5289,E1 25.0309,E2 528.6088} C_DIS
LIN {X 24.5304,Y -114.624,Z 128,A -81.2907,B 24.9568,C -1.5186,E1 25.0344,E2 527.3412} C_DIS
LIN {X 27.3303,Y -113.9888,Z 128,A -79.8876,B 24.9568,C -1.5199,E1 25.0382,E2 525.9368} C_DIS
LIN {X 30.1135,Y -113.2854,Z 128,A -78.4847,B 24.9566,C -1.5214,E1 25.042,E2 524.5326} C_DIS
LIN {X 33.1373,Y -112.4373,Z 128,A -77.0679,B 24.9568,C -1.5176,E1 25.0458,E2 523.1271} C_DIS
LIN {X 35.5615,Y -111.6954,Z 128,A -75.6729,B 24.9564,C -1.5263,E1 25.0496,E2 521.7141} C_DIS
LIN {X 38.1478,Y -110.8396,Z 128,A -74.2826,B 24.9561,C -1.5307,E1 25.0533,E2 520.316} C_DIS
LIN {X 40.8489,Y -109.8729,Z 128,A -72.788,B 24.9557,C -1.5369,E1 25.0572,E2 518.81} C_DIS
LIN {X 43.8405,Y -108.7122,Z 128,A -71.3495,B 24.956,C -1.5331,E1 25.0609,E2 517.3837} C_DIS
LIN {X 46.4124,Y -107.6396,Z 128,A -69.9623,B 24.9558,C -1.5363,E1 25.0645,E2 515.9922} C_DIS
LIN {X 48.7997,Y -106.5798,Z 128,A -68.6885,B 24.9557,C -1.5381,E1 25.0677,E2 514.7173} C_DIS
LIN {X 51.6253,Y -105.239,Z 128,A -67.0585,B 24.9553,C -1.5454,E1 25.0719,E2 513.0743} C_DIS
LIN {X 54.2352,Y -103.9178,Z 128,A -65.8543,B 24.9557,C -1.5372,E1 25.0748,E2 511.8928} C_DIS
LIN {X 56.5335,Y -102.6871,Z 128,A -64.4734,B 24.9553,C -1.5445,E1 25.0782,E2 510.4988} C_DIS
LIN {X 59.026,Y -101.275,Z 128,A -63.0764,B 24.9552,C -1.5469,E1 25.0816,E2 509.1003} C_DIS
LIN {X 61.4832,Y -99.8023,Z 128,A -61.6813,B 24.955,C -1.5493,E1 25.0849,E2 507.7039} C_DIS
LIN {X 64.1392,Y -98.115,Z 128,A -60.1506,B 24.9549,C -1.552,E1 25.0885,E2 506.1718} C_DIS
LIN {X 66.312,Y -96.6613,Z 128,A -58.7837,B 24.9545,C -1.5588,E1 25.0917,E2 504.7935} C_DIS
LIN {X 69.8406,Y -94.1433,Z 128,A -56.7699,B 24.9545,C -1.5582,E1 25.0962,E2 502.788} C_DIS
LIN {X 72.1233,Y -92.4063,Z 128,A -55.3223,B 24.9542,C -1.5635,E1 25.0995,E2 501.3333} C_DIS
LIN {X 74.8163,Y -90.2371,Z 128,A -53.6603,B 24.9541,C -1.566,E1 25.1031,E2 499.6717} C_DIS
LIN {X 77.1003,Y -88.2934,Z 128,A -52.2322,B 24.954,C -1.5675,E1 25.1061,E2 498.2455} C_DIS
LIN {X 79.2387,Y -86.3795,Z 128,A -50.8043,B 24.9537,C -1.5721,E1 25.109,E2 496.8127} C_DIS
LIN {X 81.4433,Y -84.3041,Z 128,A -49.3015,B 24.9534,C -1.5767,E1 25.1121,E2 495.3051} C_DIS
LIN {X 83.8954,Y -81.8673,Z 128,A -47.6825,B 24.9534,C -1.5775,E1 25.1152,E2 493.6911} C_DIS
LIN {X 85.9688,Y -79.6862,Z 128,A -46.227,B 24.9532,C -1.5805,E1 25.118,E2 492.2349} C_DIS
LIN {X 88.0579,Y -77.3699,Z 128,A -44.6394,B 24.9528,C -1.5875,E1 25.121,E2 490.6379} C_DIS
LIN {X 90.155,Y -74.915,Z 128,A -43.1137,B 24.9527,C -1.5892,E1 25.1237,E2 489.1152} C_DIS
LIN {X 92.0422,Y -72.5839,Z 128,A -41.6768,B 24.9525,C -1.5917,E1 25.1262,E2 487.6791} C_DIS
LIN {X 94.1754,Y -69.7971,Z 128,A -39.9651,B 24.9523,C -1.5963,E1 25.1291,E2 485.9649} C_DIS
LIN {X 95.9337,Y -67.3588,Z 128,A -38.5836,B 24.9523,C -1.5961,E1 25.1313,E2 484.5904} C_DIS
LIN {X 97.329,Y -65.3259,Z 128,A -37.2001,B 24.9515,C -1.6082,E1 25.1335,E2 483.1854} C_DIS
LIN {X 99.1703,Y -62.4952,Z 128,A -35.668,B 24.9515,C -1.6072,E1 25.1358,E2 481.6632} C_DIS
LIN {X 100.6766,Y -60.0385,Z 128,A -34.2735,B 24.9514,C -1.6106,E1 25.1379,E2 480.2678} C_DIS
LIN {X 102.1146,Y -57.5587,Z 128,A -32.8813,B 24.9512,C -1.6143,E1 25.1398,E2 478.874} C_DIS
LIN {X 103.3717,Y -55.2718,Z 128,A -31.4712,B 24.9505,C -1.6246,E1 25.1417,E2 477.447} C_DIS
LIN {X 104.6857,Y -52.7404,Z 128,A -30.1772,B 24.9505,C -1.624,E1 25.1433,E2 476.1615} C_DIS
LIN {X 105.9593,Y -50.1329,Z 128,A -28.6831,B 24.9501,C -1.632,E1 25.1451,E2 474.6566} C_DIS
LIN {X 107.1682,Y -47.4937,Z 128,A -27.4093,B 24.9503,C -1.6293,E1 25.1466,E2 473.3959} C_DIS
LIN {X 108.3959,Y -44.6174,Z 128,A -26.0034,B 24.9503,C -1.6281,E1 25.1481,E2 472.0006} C_DIS
LIN {X 109.4559,Y -41.95,Z 128,A -24.4968,B 24.9498,C -1.6375,E1 25.1496,E2 470.4801} C_DIS
LIN {X 110.4502,Y -39.2576,Z 128,A -23.1032,B 24.9495,C -1.6415,E1 25.1509,E2 469.085} C_DIS
LIN {X 111.3781,Y -36.5423,Z 128,A -21.7096,B 24.9493,C -1.6455,E1 25.1522,E2 467.6898} C_DIS
LIN {X 112.2525,Y -33.7601,Z 128,A -20.2936,B 24.949,C -1.6496,E1 25.1533,E2 466.2722} C_DIS
LIN {X 112.9788,Y -31.2484,Z 128,A -18.9301,B 24.9485,C -1.6578,E1 25.1544,E2 464.8972} C_DIS
LIN {X 113.7102,Y -28.4724,Z 128,A -17.536,B 24.9482,C -1.6619,E1 25.1553,E2 463.5015} C_DIS
LIN {X 114.3734,Y -25.679,Z 128,A -16.0606,B 24.9477,C -1.6699,E1 25.1563,E2 462.0157} C_DIS
LIN {X 115.0171,Y -22.6157,Z 128,A -14.718,B 24.948,C -1.6658,E1 25.157,E2 460.6906} C_DIS
LIN {X 115.494,Y -20.0458,Z 128,A -13.4416,B 24.9477,C -1.6699,E1 25.1576,E2 459.412} C_DIS
LIN {X 115.9897,Y -16.9347,Z 128,A -12.0329,B 24.9478,C -1.6686,E1 25.1582,E2 458.0147} C_DIS
LIN {X 116.3395,Y -14.3463,Z 128,A -10.5568,B 24.947,C -1.6824,E1 25.1587,E2 456.5147} C_DIS
LIN {X 116.6794,Y -11.2387,Z 128,A -9.2441,B 24.9473,C -1.677,E1 25.1591,E2 455.2225} C_DIS
LIN {X 116.9361,Y -8.1356,Z 128,A -7.7022,B 24.9469,C -1.683,E1 25.1595,E2 453.6757} C_DIS
LIN {X 117.0912,Y -5.4811,Z 128,A -6.3332,B 24.9464,C -1.6906,E1 25.1597,E2 452.2969} C_DIS
LIN {X 117.1855,Y -2.8709,Z 128,A -4.9353,B 24.9458,C -1.7006,E1 25.1597,E2 450.8837} C_DIS
LIN {X 117.2181,Y 0.4799,Z 128,A -3.5047,B 24.9461,C -1.696,E1 25.1597,E2 449.4726} C_DIS
LIN {X 117.1856,Y 2.8671,Z 128,A -2.2785,B 24.9457,C -1.7026,E1 25.1597,E2 448.2381} C_DIS
LIN {X 117.0803,Y 5.7338,Z 128,A -0.7707,B 24.9451,C -1.7123,E1 25.1595,E2 446.7164} C_DIS
LIN {X 116.8822,Y 8.885,Z 128,A 0.5324,B 24.9455,C -1.7057,E1 25.1593,E2 445.4365} C_DIS
LIN {X 116.6565,Y 11.4873,Z 128,A 2.0151,B 24.9446,C -1.7198,E1 25.1589,E2 443.9294} C_DIS
LIN {X 116.3075,Y 14.5937,Z 128,A 3.501,B 24.9444,C -1.7227,E1 25.1584,E2 442.4455} C_DIS
LIN {X 115.8482,Y 17.8713,Z 128,A 4.9267,B 24.9446,C -1.7186,E1 25.1578,E2 441.0378} C_DIS
LIN {X 115.2394,Y 21.4612,Z 128,A 6.8055,B 24.944,C -1.729,E1 25.1569,E2 439.1454} C_DIS
LIN {X 114.6244,Y 24.5285,Z 128,A 8.4052,B 24.9434,C -1.7373,E1 25.156,E2 437.5357} C_DIS
LIN {X 113.8854,Y 27.7542,Z 128,A 9.797,B 24.9438,C -1.7315,E1 25.1551,E2 436.1656} C_DIS
LIN {X 113.281,Y 30.1298,Z 128,A 11.0089,B 24.9435,C -1.7359,E1 25.1543,E2 434.9504} C_DIS
LIN {X 112.5091,Y 32.8952,Z 128,A 12.4038,B 24.9433,C -1.7398,E1 25.1532,E2 433.5542} C_DIS
LIN {X 111.7318,Y 35.4491,Z 128,A 13.803,B 24.9427,C -1.7483,E1 25.152,E2 432.1428} C_DIS
LIN {X 110.741,Y 38.4288,Z 128,A 15.2007,B 24.9428,C -1.7464,E1 25.1508,E2 430.7575} C_DIS
LIN {X 109.8896,Y 40.8033,Z 128,A 16.6343,B 24.942,C -1.7597,E1 25.1494,E2 429.3006} C_DIS
LIN {X 108.8397,Y 43.5271,Z 128,A 18.0754,B 24.9416,C -1.7646,E1 25.1479,E2 427.8559} C_DIS
LIN {X 107.5852,Y 46.5372,Z 128,A 19.5222,B 24.9418,C -1.7622,E1 25.1464,E2 426.4226} C_DIS
LIN {X 106.5724,Y 48.8162,Z 128,A 20.7758,B 24.9415,C -1.7674,E1 25.1449,E2 425.1636} C_DIS
LIN {X 105.2306,Y 51.6422,Z 128,A 22.2955,B 24.9412,C -1.7713,E1 25.1431,E2 423.6428} C_DIS
LIN {X 103.377,Y 55.262,Z 128,A 24.2792,B 24.9408,C -1.7767,E1 25.1405,E2 421.657} C_DIS
LIN {X 101.9841,Y 57.792,Z 128,A 25.6745,B 24.9406,C -1.7798,E1 25.1386,E2 420.2617} C_DIS
LIN {X 100.5387,Y 60.2714,Z 128,A 27.0694,B 24.9404,C -1.7832,E1 25.1366,E2 418.8658} C_DIS
LIN {X 98.8997,Y 62.9225,Z 128,A 28.5885,B 24.9401,C -1.7871,E1 25.1344,E2 417.3454} C_DIS
LIN {X 97.3234,Y 65.3341,Z 128,A 29.8748,B 24.9403,C -1.7849,E1 25.1324,E2 416.0705} C_DIS
LIN {X 95.6947,Y 67.6973,Z 128,A 31.3957,B 24.9397,C -1.7941,E1 25.1299,E2 414.5353} C_DIS
LIN {X 93.8853,Y 70.184,Z 128,A 32.9417,B 24.9393,C -1.7999,E1 25.1274,E2 412.9829} C_DIS
LIN {X 91.9138,Y 72.7465,Z 128,A 34.5112,B 24.939,C -1.8033,E1 25.1247,E2 411.413} C_DIS
LIN {X 89.7196,Y 75.439,Z 128,A 36.2606,B 24.9386,C -1.8098,E1 25.1215,E2 409.6564} C_DIS
LIN {X 87.7278,Y 77.7455,Z 128,A 37.7589,B 24.9383,C -1.8136,E1 25.1188,E2 408.1556} C_DIS
LIN {X 85.3847,Y 80.3096,Z 128,A 39.335,B 24.9385,C -1.8118,E1 25.1158,E2 406.5909} C_DIS
LIN {X 82.9771,Y 82.7969,Z 128,A 40.9414,B 24.9385,C -1.8114,E1 25.1127,E2 404.9921} C_DIS
LIN {X 80.3082,Y 85.386,Z 128,A 42.8321,B 24.938,C -1.8187,E1 25.1088,E2 403.092} C_DIS
LIN {X 77.7424,Y 87.7305,Z 128,A 44.4998,B 24.9379,C -1.8207,E1 25.1054,E2 401.4264} C_DIS
LIN {X 75.471,Y 89.6929,Z 128,A 46.0066,B 24.9375,C -1.8254,E1 25.1022,E2 399.9142} C_DIS
LIN {X 72.789,Y 91.8802,Z 128,A 47.6713,B 24.9375,C -1.8274,E1 25.0985,E2 398.2512} C_DIS
LIN {X 70.7823,Y 93.4359,Z 128,A 48.7814,B 24.9377,C -1.8235,E1 25.0961,E2 397.1542} C_DIS
LIN {X 68.6781,Y 94.9948,Z 128,A 50.2334,B 24.937,C -1.8338,E1 25.0928,E2 395.6832} C_DIS
LIN {X 66.3728,Y 96.6191,Z 128,A 51.525,B 24.937,C -1.8321,E1 25.0899,E2 394.4} C_DIS
LIN {X 63.7041,Y 98.398,Z 128,A 53.0868,B 24.937,C -1.8344,E1 25.0862,E2 392.838} C_DIS
LIN {X 61.2758,Y 99.9283,Z 128,A 54.4851,B 24.9368,C -1.8363,E1 25.0829,E2 391.4394} C_DIS
LIN {X 58.811,Y 101.3986,Z 128,A 55.8834,B 24.9367,C -1.8382,E1 25.0795,E2 390.041} C_DIS
LIN {X 56.3114,Y 102.8078,Z 128,A 57.3756,B 24.9362,C -1.8443,E1 25.0759,E2 388.5387} C_DIS
LIN {X 52.6919,Y 104.7103,Z 128,A 59.3706,B 24.9361,C -1.8468,E1 25.0709,E2 386.5434} C_DIS
LIN {X 49.8786,Y 106.0779,Z 128,A 60.6868,B 24.9366,C -1.8389,E1 25.0676,E2 385.2493} C_DIS
LIN {X 47.5014,Y 107.1649,Z 128,A 62.2054,B 24.9357,C -1.8514,E1 25.0637,E2 383.7049} C_DIS
LIN {X 44.6226,Y 108.3938,Z 128,A 63.4916,B 24.9364,C -1.8419,E1 25.0605,E2 382.4441} C_DIS
LIN {X 41.948,Y 109.4567,Z 128,A 65.0043,B 24.936,C -1.8482,E1 25.0565,E2 380.92} C_DIS
LIN {X 39.2579,Y 110.4501,Z 128,A 66.5068,B 24.9356,C -1.8541,E1 25.0525,E2 379.4067} C_DIS
LIN {X 36.531,Y 111.3817,Z 128,A 67.8019,B 24.9358,C -1.8501,E1 25.0491,E2 378.1234} C_DIS
LIN {X 34.075,Y 112.1585,Z 128,A 69.1346,B 24.9355,C -1.8544,E1 25.0455,E2 376.783} C_DIS
LIN {X 31.3747,Y 112.9432,Z 128,A 70.4616,B 24.9356,C -1.8532,E1 25.042,E2 375.461} C_DIS
LIN {X 27.9668,Y 113.8335,Z 128,A 72.1635,B 24.9356,C -1.8534,E1 25.0374,E2 373.7612} C_DIS
LIN {X 25.1875,Y 114.4806,Z 128,A 73.4701,B 24.9358,C -1.8501,E1 25.0339,E2 372.4641} C_DIS
LIN {X 22.6109,Y 115.018,Z 128,A 74.8373,B 24.9355,C -1.8544,E1 25.0301,E2 371.0886} C_DIS
LIN {X 20.0409,Y 115.4949,Z 128,A 76.1151,B 24.9355,C -1.8548,E1 25.0266,E2 369.811} C_DIS
LIN {X 16.7191,Y 116.0203,Z 128,A 77.5433,B 24.9361,C -1.8457,E1 25.0227,E2 368.4057} C_DIS
LIN {X 14.3504,Y 116.339,Z 128,A 79.0255,B 24.9352,C -1.86,E1 25.0185,E2 366.891} C_DIS
LIN {X 11.2267,Y 116.6805,Z 128,A 80.3461,B 24.9358,C -1.8506,E1 25.0149,E2 365.5935} C_DIS
LIN {X 8.0738,Y 116.9403,Z 128,A 81.9048,B 24.9358,C -1.8512,E1 25.0106,E2 364.034} C_DIS
LIN {X 5.3151,Y 117.0983,Z 128,A 83.2898,B 24.9357,C -1.8527,E1 25.0067,E2 362.646} C_DIS
LIN {X 2.8925,Y 117.1849,Z 128,A 84.6333,B 24.9352,C -1.8596,E1 25.0029,E2 361.2864} C_DIS
LIN {X 0.0214,Y 117.2206,Z 128,A 86.0451,B 24.9352,C -1.8597,E1 24.999,E2 359.8744} C_DIS
LIN {X -2.8762,Y 117.1854,Z 128,A 87.3644,B 24.9355,C -1.855,E1 24.9953,E2 358.5661} C_DIS
LIN {X -5.7441,Y 117.0799,Z 128,A 88.8613,B 24.9352,C -1.8587,E1 24.9911,E2 357.0602} C_DIS
LIN {X -8.8642,Y 116.8839,Z 128,A 90.3334,B 24.9355,C -1.8556,E1 24.987,E2 355.5948} C_DIS
LIN {X -11.4835,Y 116.6568,Z 128,A 91.6828,B 24.9353,C -1.8578,E1 24.9833,E2 354.2396} C_DIS
LIN {X -14.6065,Y 116.3058,Z 128,A 93.0074,B 24.936,C -1.8477,E1 24.9796,E2 352.9382} C_DIS
LIN {X -17.4497,Y 115.9134,Z 128,A 94.526,B 24.9357,C -1.8518,E1 24.9754,E2 351.4086} C_DIS
LIN {X -20.0292,Y 115.4968,Z 128,A 95.8065,B 24.9357,C -1.851,E1 24.9719,E2 350.1288} C_DIS
LIN {X -23.108,Y 114.9192,Z 128,A 97.4472,B 24.9355,C -1.8545,E1 24.9674,E2 348.4777} C_DIS
LIN {X -25.8996,Y 114.3225,Z 128,A 98.7518,B 24.9359,C -1.8493,E1 24.9638,E2 347.184} C_DIS
LIN {X -28.4808,Y 113.7081,Z 128,A 100.1334,B 24.9357,C -1.8517,E1 24.9601,E2 345.7947} C_DIS
LIN {X -31.257,Y 112.9765,Z 128,A 101.5517,B 24.9357,C -1.8509,E1 24.9563,E2 344.3762} C_DIS
LIN {X -34.047,Y 112.1672,Z 128,A 102.8619,B 24.9362,C -1.8446,E1 24.9528,E2 343.0788} C_DIS
LIN {X -36.7639,Y 111.3064,Z 128,A 104.2758,B 24.9362,C -1.8438,E1 24.949,E2 341.6642} C_DIS
LIN {X -39.4581,Y 110.3798,Z 128,A 105.6608,B 24.9364,C -1.8417,E1 24.9454,E2 340.2814} C_DIS
LIN {X -42.3541,Y 109.3005,Z 128,A 107.0963,B 24.9368,C -1.8365,E1 24.9417,E2 338.8553} C_DIS
LIN {X -45.0958,Y 108.1978,Z 128,A 108.6497,B 24.9366,C -1.8391,E1 24.9376,E2 337.2922} C_DIS
LIN {X -47.7366,Y 107.0589,Z 128,A 109.9212,B 24.9371,C -1.8313,E1 24.9344,E2 336.0364} C_DIS
LIN {X -50.1124,Y 105.969,Z 128,A 111.4109,B 24.9367,C -1.8383,E1 24.9306,E2 334.5262} C_DIS
LIN {X -52.9461,Y 104.5805,Z 128,A 112.8623,B 24.9371,C -1.8319,E1 24.927,E2 333.0861} C_DIS
LIN {X -55.2585,Y 103.3789,Z 128,A 114.143,B 24.9372,C -1.8301,E1 24.9238,E2 331.8063} C_DIS
LIN {X -57.7663,Y 101.9987,Z 128,A 115.5479,B 24.9374,C -1.8278,E1 24.9204,E2 330.4026} C_DIS
LIN {X -60.2385,Y 100.5583,Z 128,A 116.9519,B 24.9375,C -1.8255,E1 24.917,E2 328.9998} C_DIS
LIN {X -62.6721,Y 99.0598,Z 128,A 118.4501,B 24.9375,C -1.8272,E1 24.9135,E2 327.493} C_DIS
LIN {X -65.4463,Y 97.2475,Z 128,A 120.0017,B 24.9378,C -1.8211,E1 24.9099,E2 325.9507} C_DIS
LIN {X -67.7179,Y 95.68,Z 128,A 121.3342,B 24.9381,C -1.8177,E1 24.9068,E2 324.6219} C_DIS
LIN {X -69.8312,Y 94.1504,Z 128,A 122.6154,B 24.9382,C -1.8152,E1 24.904,E2 323.3419} C_DIS
LIN {X -72.1118,Y 92.4153,Z 128,A 124.0716,B 24.9382,C -1.8146,E1 24.9007,E2 321.8819} C_DIS
LIN {X -74.7705,Y 90.2751,Z 128,A 125.7477,B 24.9385,C -1.8112,E1 24.8971,E2 320.2075} C_DIS
LIN {X -77.1052,Y 88.2891,Z 128,A 127.209,B 24.9388,C -1.8063,E1 24.894,E2 318.7523} C_DIS
LIN {X -79.2528,Y 86.3665,Z 128,A 128.6469,B 24.939,C -1.8042,E1 24.891,E2 317.3135} C_DIS
LIN {X -81.4301,Y 84.3169,Z 128,A 130.1549,B 24.939,C -1.8026,E1 24.888,E2 315.803} C_DIS
LIN {X -84.1812,Y 81.5708,Z 128,A 132.0529,B 24.9394,C -1.7979,E1 24.8843,E2 313.9082} C_DIS
LIN {X -86.3754,Y 79.2431,Z 128,A 133.5724,B 24.9398,C -1.7921,E1 24.8814,E2 312.3959} C_DIS
LIN {X -88.3702,Y 77.0123,Z 128,A 135.1076,B 24.9398,C -1.7913,E1 24.8786,E2 310.8556} C_DIS
LIN {X -90.6789,Y 74.2826,Z 128,A 136.9358,B 24.9399,C -1.7901,E1 24.8753,E2 309.0219} C_DIS
LIN {X -92.8486,Y 71.5495,Z 128,A 138.3718,B 24.941,C -1.7743,E1 24.8729,E2 307.6169} C_DIS
LIN {X -95.0033,Y 68.6663,Z 128,A 140.3831,B 24.9406,C -1.7799,E1 24.8695,E2 305.5824} C_DIS
LIN {X -96.6548,Y 66.3215,Z 128,A 141.698,B 24.9411,C -1.7724,E1 24.8674,E2 304.279} C_DIS
LIN {X -98.5535,Y 63.462,Z 128,A 143.265,B 24.9417,C -1.763,E1 24.865,E2 302.7264} C_DIS
LIN {X -99.8324,Y 61.4336,Z 128,A 144.675,B 24.9413,C -1.7695,E1 24.8629,E2 301.2937} C_DIS
LIN {X -102.1255,Y 57.5393,Z 128,A 146.7869,B 24.942,C -1.759,E1 24.86,E2 299.1958} C_DIS
LIN {X -103.3828,Y 55.2511,Z 128,A 148.1349,B 24.942,C -1.7582,E1 24.8582,E2 297.8426} C_DIS
LIN {X -104.7037,Y 52.7051,Z 128,A 149.5792,B 24.9422,C -1.7557,E1 24.8564,E2 296.3965} C_DIS
LIN {X -106.0703,Y 49.8949,Z 128,A 151.1183,B 24.9425,C -1.7516,E1 24.8545,E2 294.8588} C_DIS
LIN {X -107.8603,Y 45.8967,Z 128,A 153.2621,B 24.9429,C -1.7452,E1 24.8521,E2 292.7187} C_DIS
LIN {X -109.457,Y 41.9472,Z 128,A 155.2823,B 24.9435,C -1.7361,E1 24.8501,E2 290.7086} C_DIS
LIN {X -110.46,Y 39.2296,Z 128,A 156.697,B 24.9438,C -1.7316,E1 24.8487,E2 289.2967} C_DIS
LIN {X -111.3864,Y 36.5166,Z 128,A 158.1079,B 24.9441,C -1.7276,E1 24.8475,E2 287.8874} C_DIS
LIN {X -112.1732,Y 34.0276,Z 128,A 159.4899,B 24.9441,C -1.7279,E1 24.8463,E2 286.4966} C_DIS
LIN {X -112.9718,Y 31.2738,Z 128,A 160.8978,B 24.9443,C -1.7237,E1 24.8453,E2 285.0906} C_DIS
LIN {X -113.7028,Y 28.5018,Z 128,A 162.3052,B 24.9446,C -1.7194,E1 24.8443,E2 283.6851} C_DIS
LIN {X -114.3936,Y 25.5864,Z 128,A 163.8384,B 24.9447,C -1.7176,E1 24.8433,E2 282.1474} C_DIS
LIN {X -115.0203,Y 22.599,Z 128,A 165.1925,B 24.9454,C -1.707,E1 24.8426,E2 280.8103} C_DIS
LIN {X -115.4968,Y 20.0293,Z 128,A 166.4781,B 24.9456,C -1.7032,E1 24.842,E2 279.5263} C_DIS
LIN {X -116.0173,Y 16.7398,Z 128,A 167.9157,B 24.9465,C -1.6901,E1 24.8414,E2 278.1114} C_DIS
LIN {X -116.3394,Y 14.3468,Z 128,A 169.4043,B 24.9459,C -1.6989,E1 24.8408,E2 276.5929} C_DIS
LIN {X -116.7047,Y 10.9656,Z 128,A 171.0318,B 24.9463,C -1.6921,E1 24.8404,E2 274.9719} C_DIS
LIN {X -117.0149,Y 6.9201,Z 128,A 172.9784,B 24.9469,C -1.6841,E1 24.84,E2 273.0327} C_DIS
LIN {X -117.1493,Y 4.0523,Z 128,A 174.276,B 24.9474,C -1.6751,E1 24.8399,E2 271.7487} C_DIS
LIN {X -117.2144,Y 1.0533,Z 128,A 175.8771,B 24.9474,C -1.6759,E1 24.8398,E2 270.1361} C_DIS
LIN {X -117.2017,Y -1.9932,Z 128,A 177.3947,B 24.9476,C -1.6722,E1 24.8398,E2 268.618} C_DIS
LIN {X -117.0791,Y -5.7599,Z 128,A 179.3194,B 24.9478,C -1.6696,E1 24.8401,E2 266.6879} C_DIS
LIN {X -116.8822,Y -8.8849,Z 128,A -179.3503,B 24.9486,C -1.6564,E1 24.8403,E2 265.3811} C_DIS
LIN {X -116.6563,Y -11.489,Z 128,A -177.8523,B 24.9483,C -1.6614,E1 24.8407,E2 263.8624} C_DIS
LIN {X -116.2685,Y -14.8942,Z 128,A -176.4996,B 24.9494,C -1.6427,E1 24.8411,E2 262.5461} C_DIS
LIN {X -115.9117,Y -17.4601,Z 128,A -174.9873,B 24.9491,C -1.6488,E1 24.8417,E2 261.0102} C_DIS
LIN {X -115.4949,Y -20.0406,Z 128,A -173.5507,B 24.9489,C -1.6513,E1 24.8424,E2 259.5592} C_DIS
LIN {X -114.9465,Y -22.9749,Z 128,A -172.1679,B 24.9494,C -1.6435,E1 24.8432,E2 258.1867} C_DIS
LIN {X -114.2638,Y -26.1537,Z 128,A -170.7204,B 24.95,C -1.6327,E1 24.844,E2 256.7566} C_DIS
LIN {X -113.7185,Y -28.4385,Z 128,A -169.4053,B 24.9498,C -1.636,E1 24.8449,E2 255.4258} C_DIS
LIN {X -113.0026,Y -31.1604,Z 128,A -168.062,B 24.9502,C -1.6304,E1 24.8459,E2 254.088} C_DIS
LIN {X -112.1707,Y -34.0357,Z 128,A -166.6191,B 24.9505,C -1.6251,E1 24.847,E2 252.6495} C_DIS
LIN {X -111.2968,Y -36.7925,Z 128,A -165.2048,B 24.9508,C -1.6208,E1 24.8482,E2 251.2372} C_DIS
LIN {X -110.2179,Y -39.9034,Z 128,A -163.7699,B 24.9515,C -1.6088,E1 24.8496,E2 249.823} C_DIS
LIN {X -109.1704,Y -42.6853,Z 128,A -162.0668,B 24.9511,C -1.6149,E1 24.8513,E2 248.0958} C_DIS
LIN {X -108.1959,Y -45.1002,Z 128,A -160.8322,B 24.9515,C -1.6095,E1 24.8526,E2 246.867} C_DIS
LIN {X -107.0589,Y -47.7366,Z 128,A -159.533,B 24.952,C -1.6011,E1 24.854,E2 245.5808} C_DIS
LIN {X -105.9562,Y -50.1393,Z 128,A -158.0269,B 24.9517,C -1.6063,E1 24.8558,E2 244.054} C_DIS
LIN {X -104.5871,Y -52.9334,Z 128,A -156.5923,B 24.9521,C -1.5984,E1 24.8576,E2 242.6305} C_DIS
LIN {X -103.3883,Y -55.2406,Z 128,A -155.3099,B 24.9523,C -1.5953,E1 24.8593,E2 241.3486} C_DIS
LIN {X -102.0131,Y -57.7406,Z 128,A -153.9044,B 24.9525,C -1.592,E1 24.8612,E2 239.9437} C_DIS
LIN {X -100.4147,Y -60.4755,Z 128,A -152.4587,B 24.953,C -1.5835,E1 24.8632,E2 238.5107} C_DIS
LIN {X -99.0352,Y -62.7115,Z 128,A -150.9616,B 24.9527,C -1.5891,E1 24.8655,E2 236.9928} C_DIS
LIN {X -97.3127,Y -65.35,Z 128,A -149.6252,B 24.9534,C -1.5765,E1 24.8675,E2 235.6797} C_DIS
LIN {X -95.564,Y -67.8805,Z 128,A -148.0738,B 24.9535,C -1.5747,E1 24.87,E2 234.125} C_DIS
LIN {X -94.1576,Y -69.8215,Z 128,A -146.8197,B 24.9535,C -1.5752,E1 24.8721,E2 232.8635} C_DIS
LIN {X -92.4234,Y -72.1012,Z 128,A -145.2768,B 24.9534,C -1.5778,E1 24.8747,E2 231.307} C_DIS
LIN {X -90.229,Y -74.8259,Z 128,A -143.6651,B 24.9538,C -1.5696,E1 24.8775,E2 229.7074} C_DIS
LIN {X -88.1485,Y -77.2662,Z 128,A -142.0596,B 24.954,C -1.5676,E1 24.8805,E2 228.0994} C_DIS
LIN {X -85.8061,Y -79.8615,Z 128,A -140.2708,B 24.954,C -1.5671,E1 24.8839,E2 226.3039} C_DIS
LIN {X -83.3932,Y -82.3757,Z 128,A -138.6635,B 24.9544,C -1.5593,E1 24.887,E2 224.7082} C_DIS
LIN {X -80.9253,Y -84.8034,Z 128,A -136.9401,B 24.9546,C -1.5571,E1 24.8904,E2 222.983} C_DIS
Enddeposition()
END
